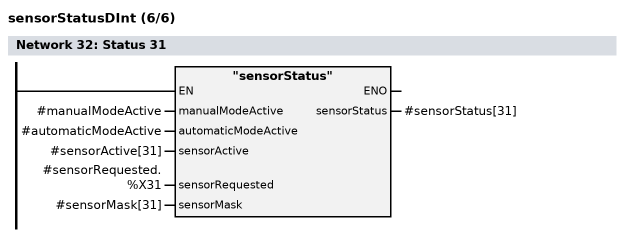
   RUNG wire#powerrail
      "sensorStatus"(manualModeActive := #manualModeActive, automaticModeActive := #automaticModeActive, sensorActive := #sensorActive[31], sensorRequested := #sensorRequested.%X31, sensorMask := #sensorMask[31], sensorStatus => #sensorStatus[31])
   END_RUNG
   // the same network as SCL:
   "sensorStatus"(manualModeActive := #manualModeActive,
                  automaticModeActive := #automaticModeActive,
                  sensorActive := #sensorActive[31],
                  sensorRequested := #sensorRequested.%X31,
                  sensorMask := #sensorMask[31],
                  sensorStatus => #sensorStatus[31]);
END_REGION
END_FUNCTION

FUNCTION "sensorStatus" : Void   // FC36, LAD
{ S7_Optimized_Access := 'TRUE' }
VERSION : 0.1
// stored: AutoNumber true, IsIECCheckEnabled false, SetENOAutomatically false, UDAEnableTagReadback false
   VAR_INPUT
      manualModeActive : Bool;
      automaticModeActive : Bool;
      sensorActive : Bool;
      sensorRequested : Bool;
      sensorMask : Bool;
   END_VAR
   VAR_OUTPUT
      sensorStatus : Int;
   END_VAR
   VAR_TEMP
      localMask : Bool;
   END_VAR
BEGIN

REGION Network 1
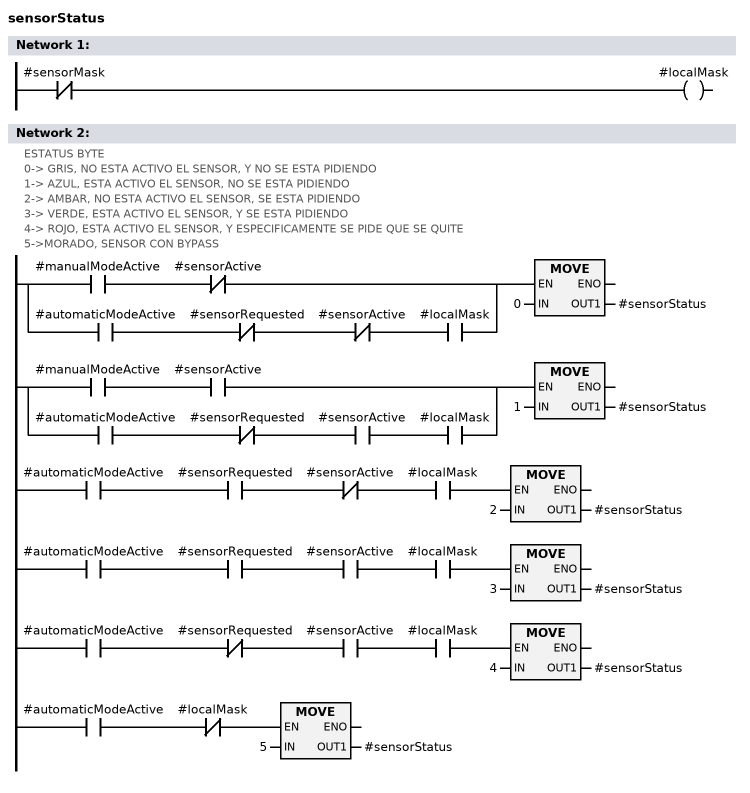
   RUNG wire#powerrail
      I_Contact( #sensorMask )
      Coil( #localMask )
   END_RUNG
   // the same network as SCL:
   #localMask := NOT #sensorMask;
END_REGION

REGION Network 2
   // ESTATUS BYTE
   // 0-> GRIS, NO ESTA ACTIVO EL SENSOR, Y NO SE ESTA PIDIENDO
   // 1-> AZUL, ESTA ACTIVO EL SENSOR, NO SE ESTA PIDIENDO
   // 2-> AMBAR, NO ESTA ACTIVO EL SENSOR, SE ESTA PIDIENDO
   // 3-> VERDE, ESTA ACTIVO EL SENSOR, Y SE ESTA PIDIENDO
   // 4-> ROJO, ESTA ACTIVO EL SENSOR, Y ESPECIFICAMENTE SE PIDE QUE SE QUITE
   // 5->MORADO, SENSOR CON BYPASS
   RUNG wire#powerrail
      Contact( #manualModeActive )
      I_Contact( #sensorActive )
      wire#w1
      Move(in := 0, out1 => #sensorStatus)
   END_RUNG
   RUNG wire#powerrail
      Contact( #automaticModeActive )
      I_Contact( #sensorRequested )
      I_Contact( #sensorActive )
      Contact( #localMask )
   END_RUNG wire#w1
   RUNG wire#powerrail
      Contact( #manualModeActive )
      Contact( #sensorActive )
      wire#w2
      Move(in := 1, out1 => #sensorStatus)
   END_RUNG
   RUNG wire#powerrail
      Contact( #automaticModeActive )
      I_Contact( #sensorRequested )
      Contact( #sensorActive )
      Contact( #localMask )
   END_RUNG wire#w2
   RUNG wire#powerrail
      Contact( #automaticModeActive )
      Contact( #sensorRequested )
      I_Contact( #sensorActive )
      Contact( #localMask )
      Move(in := 2, out1 => #sensorStatus)
   END_RUNG
   RUNG wire#powerrail
      Contact( #automaticModeActive )
      Contact( #sensorRequested )
      Contact( #sensorActive )
      Contact( #localMask )
      Move(in := 3, out1 => #sensorStatus)
   END_RUNG
   RUNG wire#powerrail
      Contact( #automaticModeActive )
      I_Contact( #sensorRequested )
      Contact( #sensorActive )
      Contact( #localMask )
      Move(in := 4, out1 => #sensorStatus)
   END_RUNG
   RUNG wire#powerrail
      Contact( #automaticModeActive )
      I_Contact( #localMask )
      Move(in := 5, out1 => #sensorStatus)
   END_RUNG
   // the same network as SCL:
   IF (#manualModeActive AND NOT #sensorActive) OR (#automaticModeActive AND NOT #sensorRequested AND NOT #sensorActive AND #localMask) THEN
       #sensorStatus := 0;
   END_IF;
   IF (#manualModeActive AND #sensorActive) OR (#automaticModeActive AND NOT #sensorRequested AND #sensorActive AND #localMask) THEN
       #sensorStatus := 1;
   END_IF;
   IF #automaticModeActive AND #sensorRequested AND NOT #sensorActive AND #localMask THEN
       #sensorStatus := 2;
   END_IF;
   IF #automaticModeActive AND #sensorRequested AND #sensorActive AND #localMask THEN
       #sensorStatus := 3;
   END_IF;
   IF #automaticModeActive AND NOT #sensorRequested AND #sensorActive AND #localMask THEN
       #sensorStatus := 4;
   END_IF;
   IF #automaticModeActive AND NOT #localMask THEN #sensorStatus := 5; END_IF;
END_REGION
END_FUNCTION

FUNCTION "cylinderControl" : Void   // FC9, LAD
{ S7_Optimized_Access := 'TRUE' }
VERSION : 0.1
// stored: AutoNumber true, IsIECCheckEnabled false, SetENOAutomatically false, UDAEnableTagReadback false
   VAR_TEMP
      enableCylinders : Bool;
   END_VAR
   VAR_TEMP   // added for the SCL form of the ladder/FBD networks
      _w1 : Bool;
      _w2 : Bool;
   END_VAR
BEGIN

REGION Network 1
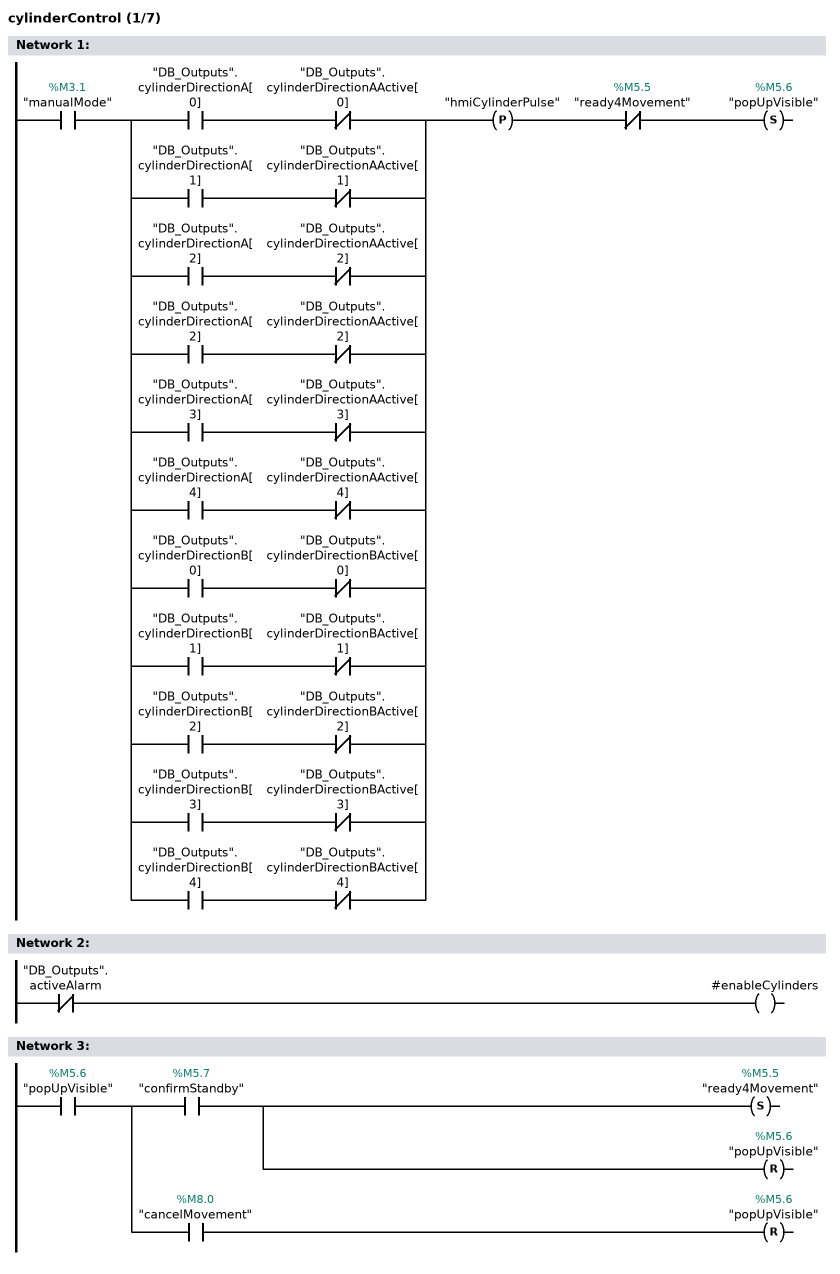
   RUNG wire#powerrail
      Contact( "manualMode" )
      wire#w1
      Contact( "DB_Outputs".cylinderDirectionA[0] )
      I_Contact( "DB_Outputs".cylinderDirectionAActive[0] )
      wire#w2
      P_Trig( "hmiCylinderPulse" )
      I_Contact( "ready4Movement" )
      S_Coil( "popUpVisible" )
   END_RUNG
   RUNG wire#w1
      Contact( "DB_Outputs".cylinderDirectionA[1] )
      I_Contact( "DB_Outputs".cylinderDirectionAActive[1] )
   END_RUNG wire#w2
   RUNG wire#w1
      Contact( "DB_Outputs".cylinderDirectionA[2] )
      I_Contact( "DB_Outputs".cylinderDirectionAActive[2] )
   END_RUNG wire#w2
   RUNG wire#w1
      Contact( "DB_Outputs".cylinderDirectionA[2] )
      I_Contact( "DB_Outputs".cylinderDirectionAActive[2] )
   END_RUNG wire#w2
   RUNG wire#w1
      Contact( "DB_Outputs".cylinderDirectionA[3] )
      I_Contact( "DB_Outputs".cylinderDirectionAActive[3] )
   END_RUNG wire#w2
   RUNG wire#w1
      Contact( "DB_Outputs".cylinderDirectionA[4] )
      I_Contact( "DB_Outputs".cylinderDirectionAActive[4] )
   END_RUNG wire#w2
   RUNG wire#w1
      Contact( "DB_Outputs".cylinderDirectionB[0] )
      I_Contact( "DB_Outputs".cylinderDirectionBActive[0] )
   END_RUNG wire#w2
   RUNG wire#w1
      Contact( "DB_Outputs".cylinderDirectionB[1] )
      I_Contact( "DB_Outputs".cylinderDirectionBActive[1] )
   END_RUNG wire#w2
   RUNG wire#w1
      Contact( "DB_Outputs".cylinderDirectionB[2] )
      I_Contact( "DB_Outputs".cylinderDirectionBActive[2] )
   END_RUNG wire#w2
   RUNG wire#w1
      Contact( "DB_Outputs".cylinderDirectionB[3] )
      I_Contact( "DB_Outputs".cylinderDirectionBActive[3] )
   END_RUNG wire#w2
   RUNG wire#w1
      Contact( "DB_Outputs".cylinderDirectionB[4] )
      I_Contact( "DB_Outputs".cylinderDirectionBActive[4] )
   END_RUNG wire#w2
   // the same network as SCL:
   #_w1 := "manualMode" AND (("DB_Outputs".cylinderDirectionA[0] AND NOT "DB_Outputs".cylinderDirectionAActive[0]) OR ("DB_Outputs".cylinderDirectionA[1] AND NOT "DB_Outputs".cylinderDirectionAActive[1]) OR ("DB_Outputs".cylinderDirectionA[2] AND NOT "DB_Outputs".cylinderDirectionAActive[2]) OR ("DB_Outputs".cylinderDirectionA[2] AND NOT "DB_Outputs".cylinderDirectionAActive[2]) OR ("DB_Outputs".cylinderDirectionA[3] AND NOT "DB_Outputs".cylinderDirectionAActive[3]) OR ("DB_Outputs".cylinderDirectionA[4] AND NOT "DB_Outputs".cylinderDirectionAActive[4]) OR ("DB_Outputs".cylinderDirectionB[0] AND NOT "DB_Outputs".cylinderDirectionBActive[0]) OR ("DB_Outputs".cylinderDirectionB[1] AND NOT "DB_Outputs".cylinderDirectionBActive[1]) OR ("DB_Outputs".cylinderDirectionB[2] AND NOT "DB_Outputs".cylinderDirectionBActive[2]) OR ("DB_Outputs".cylinderDirectionB[3] AND NOT "DB_Outputs".cylinderDirectionBActive[3]) OR ("DB_Outputs".cylinderDirectionB[4] AND NOT "DB_Outputs".cylinderDirectionBActive[4]));
   #_w2 := #_w1 AND NOT "hmiCylinderPulse";   // rising edge
   "hmiCylinderPulse" := #_w1;
   IF #_w2 AND NOT "ready4Movement" THEN "popUpVisible" := TRUE; END_IF;
END_REGION

REGION Network 2
   RUNG wire#powerrail
      I_Contact( "DB_Outputs".activeAlarm )
      Coil( #enableCylinders )
   END_RUNG
   // the same network as SCL:
   #enableCylinders := NOT "DB_Outputs".activeAlarm;
END_REGION

REGION Network 3
   RUNG wire#powerrail
      Contact( "popUpVisible" )
      wire#w1
      Contact( "confirmStandby" )
      wire#w2
      S_Coil( "ready4Movement" )
   END_RUNG
   RUNG wire#w2
      R_Coil( "popUpVisible" )
   END_RUNG
   RUNG wire#w1
      Contact( "cancelMovement" )
      R_Coil( "popUpVisible" )
   END_RUNG
   // the same network as SCL:
   IF "popUpVisible" AND "confirmStandby" THEN "ready4Movement" := TRUE; END_IF;
   #_w1 := "popUpVisible";
   IF "popUpVisible" AND "confirmStandby" THEN "popUpVisible" := FALSE; END_IF;
   IF #_w1 AND "cancelMovement" THEN "popUpVisible" := FALSE; END_IF;
END_REGION

REGION Network 4: EXT CYL 1.- LEFT TOOLING LOCK EXTENDED
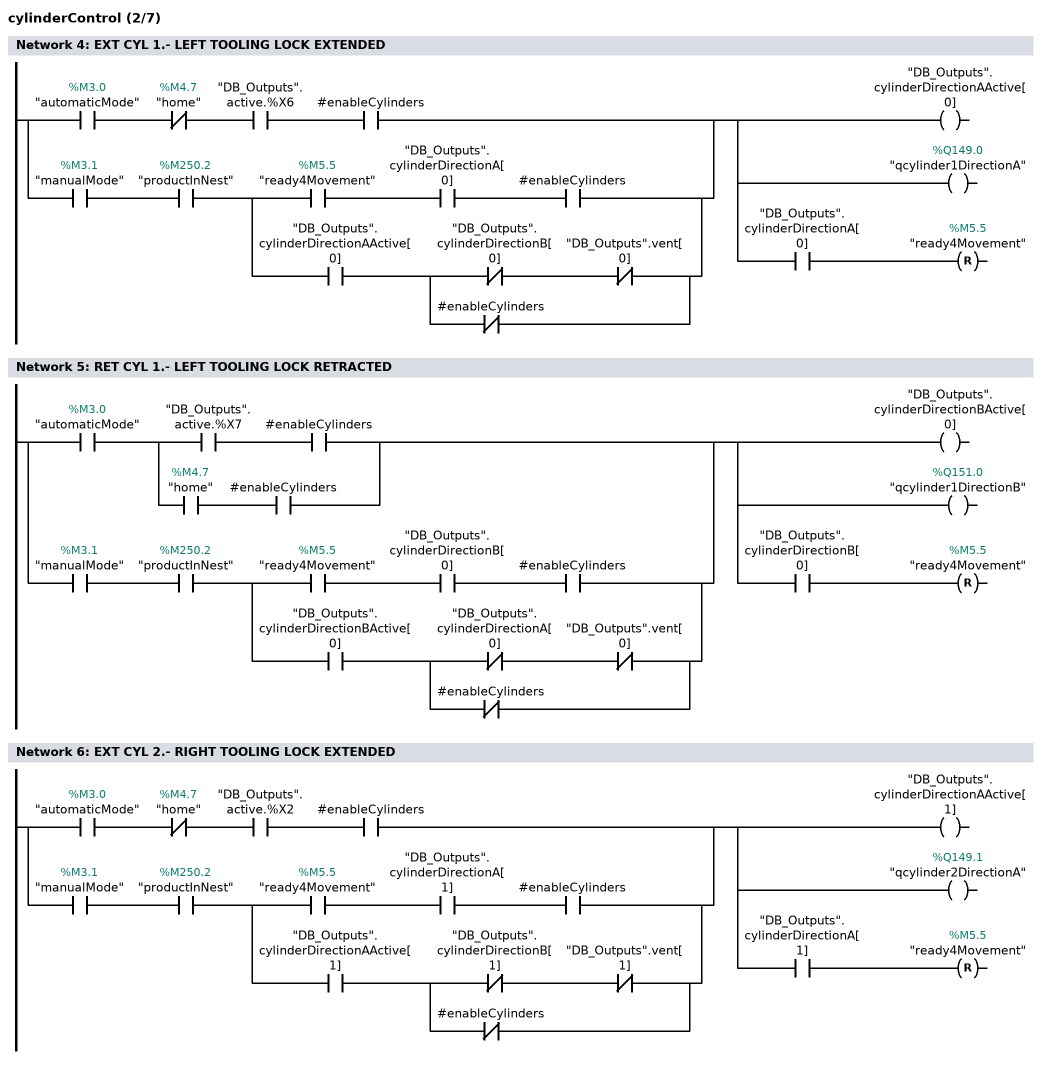
   RUNG wire#powerrail
      Contact( "automaticMode" )
      I_Contact( "home" )
      Contact( "DB_Outputs".active.%X6 )
      Contact( #enableCylinders )
      wire#w1
      Coil( "DB_Outputs".cylinderDirectionAActive[0] )
   END_RUNG
   RUNG wire#powerrail
      Contact( "manualMode" )
      Contact( "productInNest" )
      wire#w2
      Contact( "ready4Movement" )
      Contact( "DB_Outputs".cylinderDirectionA[0] )
      Contact( #enableCylinders )
   END_RUNG wire#w1
   RUNG wire#w2
      Contact( "DB_Outputs".cylinderDirectionAActive[0] )
      wire#w3
      I_Contact( "DB_Outputs".cylinderDirectionB[0] )
      I_Contact( "DB_Outputs".vent[0] )
   END_RUNG wire#w1
   RUNG wire#w3
      I_Contact( #enableCylinders )
   END_RUNG wire#w1
   RUNG wire#w1
      Coil( "qcylinder1DirectionA" )
   END_RUNG
   RUNG wire#w1
      Contact( "DB_Outputs".cylinderDirectionA[0] )
      R_Coil( "ready4Movement" )
   END_RUNG
   // the same network as SCL:
   #_w1 := ("automaticMode" AND NOT "home" AND "DB_Outputs".active.%X6 AND #enableCylinders) OR ("manualMode" AND "productInNest" AND (("ready4Movement" AND "DB_Outputs".cylinderDirectionA[0] AND #enableCylinders) OR ("DB_Outputs".cylinderDirectionAActive[0] AND ((NOT "DB_Outputs".cylinderDirectionB[0] AND NOT "DB_Outputs".vent[0]) OR NOT #enableCylinders))));
   "DB_Outputs".cylinderDirectionAActive[0] := ("automaticMode" AND NOT "home" AND "DB_Outputs".active.%X6 AND #enableCylinders) OR ("manualMode" AND "productInNest" AND (("ready4Movement" AND "DB_Outputs".cylinderDirectionA[0] AND #enableCylinders) OR ("DB_Outputs".cylinderDirectionAActive[0] AND ((NOT "DB_Outputs".cylinderDirectionB[0] AND NOT "DB_Outputs".vent[0]) OR NOT #enableCylinders))));
   "qcylinder1DirectionA" := #_w1;
   IF #_w1 AND "DB_Outputs".cylinderDirectionA[0] THEN "ready4Movement" := FALSE; END_IF;
END_REGION

REGION Network 5: RET CYL 1.- LEFT TOOLING LOCK RETRACTED
   RUNG wire#powerrail
      Contact( "automaticMode" )
      wire#w1
      Contact( "DB_Outputs".active.%X7 )
      Contact( #enableCylinders )
      wire#w2
      Coil( "DB_Outputs".cylinderDirectionBActive[0] )
   END_RUNG
   RUNG wire#w1
      Contact( "home" )
      Contact( #enableCylinders )
   END_RUNG wire#w2
   RUNG wire#powerrail
      Contact( "manualMode" )
      Contact( "productInNest" )
      wire#w3
      Contact( "ready4Movement" )
      Contact( "DB_Outputs".cylinderDirectionB[0] )
      Contact( #enableCylinders )
   END_RUNG wire#w2
   RUNG wire#w3
      Contact( "DB_Outputs".cylinderDirectionBActive[0] )
      wire#w4
      I_Contact( "DB_Outputs".cylinderDirectionA[0] )
      I_Contact( "DB_Outputs".vent[0] )
   END_RUNG wire#w2
   RUNG wire#w4
      I_Contact( #enableCylinders )
   END_RUNG wire#w2
   RUNG wire#w2
      Coil( "qcylinder1DirectionB" )
   END_RUNG
   RUNG wire#w2
      Contact( "DB_Outputs".cylinderDirectionB[0] )
      R_Coil( "ready4Movement" )
   END_RUNG
   // the same network as SCL:
   #_w1 := ("automaticMode" AND (("DB_Outputs".active.%X7 AND #enableCylinders) OR ("home" AND #enableCylinders))) OR ("manualMode" AND "productInNest" AND (("ready4Movement" AND "DB_Outputs".cylinderDirectionB[0] AND #enableCylinders) OR ("DB_Outputs".cylinderDirectionBActive[0] AND ((NOT "DB_Outputs".cylinderDirectionA[0] AND NOT "DB_Outputs".vent[0]) OR NOT #enableCylinders))));
   "DB_Outputs".cylinderDirectionBActive[0] := ("automaticMode" AND (("DB_Outputs".active.%X7 AND #enableCylinders) OR ("home" AND #enableCylinders))) OR ("manualMode" AND "productInNest" AND (("ready4Movement" AND "DB_Outputs".cylinderDirectionB[0] AND #enableCylinders) OR ("DB_Outputs".cylinderDirectionBActive[0] AND ((NOT "DB_Outputs".cylinderDirectionA[0] AND NOT "DB_Outputs".vent[0]) OR NOT #enableCylinders))));
   "qcylinder1DirectionB" := #_w1;
   IF #_w1 AND "DB_Outputs".cylinderDirectionB[0] THEN "ready4Movement" := FALSE; END_IF;
END_REGION

REGION Network 6: EXT CYL 2.- RIGHT TOOLING LOCK EXTENDED
   RUNG wire#powerrail
      Contact( "automaticMode" )
      I_Contact( "home" )
      Contact( "DB_Outputs".active.%X2 )
      Contact( #enableCylinders )
      wire#w1
      Coil( "DB_Outputs".cylinderDirectionAActive[1] )
   END_RUNG
   RUNG wire#powerrail
      Contact( "manualMode" )
      Contact( "productInNest" )
      wire#w2
      Contact( "ready4Movement" )
      Contact( "DB_Outputs".cylinderDirectionA[1] )
      Contact( #enableCylinders )
   END_RUNG wire#w1
   RUNG wire#w2
      Contact( "DB_Outputs".cylinderDirectionAActive[1] )
      wire#w3
      I_Contact( "DB_Outputs".cylinderDirectionB[1] )
      I_Contact( "DB_Outputs".vent[1] )
   END_RUNG wire#w1
   RUNG wire#w3
      I_Contact( #enableCylinders )
   END_RUNG wire#w1
   RUNG wire#w1
      Coil( "qcylinder2DirectionA" )
   END_RUNG
   RUNG wire#w1
      Contact( "DB_Outputs".cylinderDirectionA[1] )
      R_Coil( "ready4Movement" )
   END_RUNG
   // the same network as SCL:
   #_w1 := ("automaticMode" AND NOT "home" AND "DB_Outputs".active.%X2 AND #enableCylinders) OR ("manualMode" AND "productInNest" AND (("ready4Movement" AND "DB_Outputs".cylinderDirectionA[1] AND #enableCylinders) OR ("DB_Outputs".cylinderDirectionAActive[1] AND ((NOT "DB_Outputs".cylinderDirectionB[1] AND NOT "DB_Outputs".vent[1]) OR NOT #enableCylinders))));
   "DB_Outputs".cylinderDirectionAActive[1] := ("automaticMode" AND NOT "home" AND "DB_Outputs".active.%X2 AND #enableCylinders) OR ("manualMode" AND "productInNest" AND (("ready4Movement" AND "DB_Outputs".cylinderDirectionA[1] AND #enableCylinders) OR ("DB_Outputs".cylinderDirectionAActive[1] AND ((NOT "DB_Outputs".cylinderDirectionB[1] AND NOT "DB_Outputs".vent[1]) OR NOT #enableCylinders))));
   "qcylinder2DirectionA" := #_w1;
   IF #_w1 AND "DB_Outputs".cylinderDirectionA[1] THEN "ready4Movement" := FALSE; END_IF;
END_REGION

REGION Network 7: RET CYL 2.- RIGHT TOOLING LOCK RETRACTED
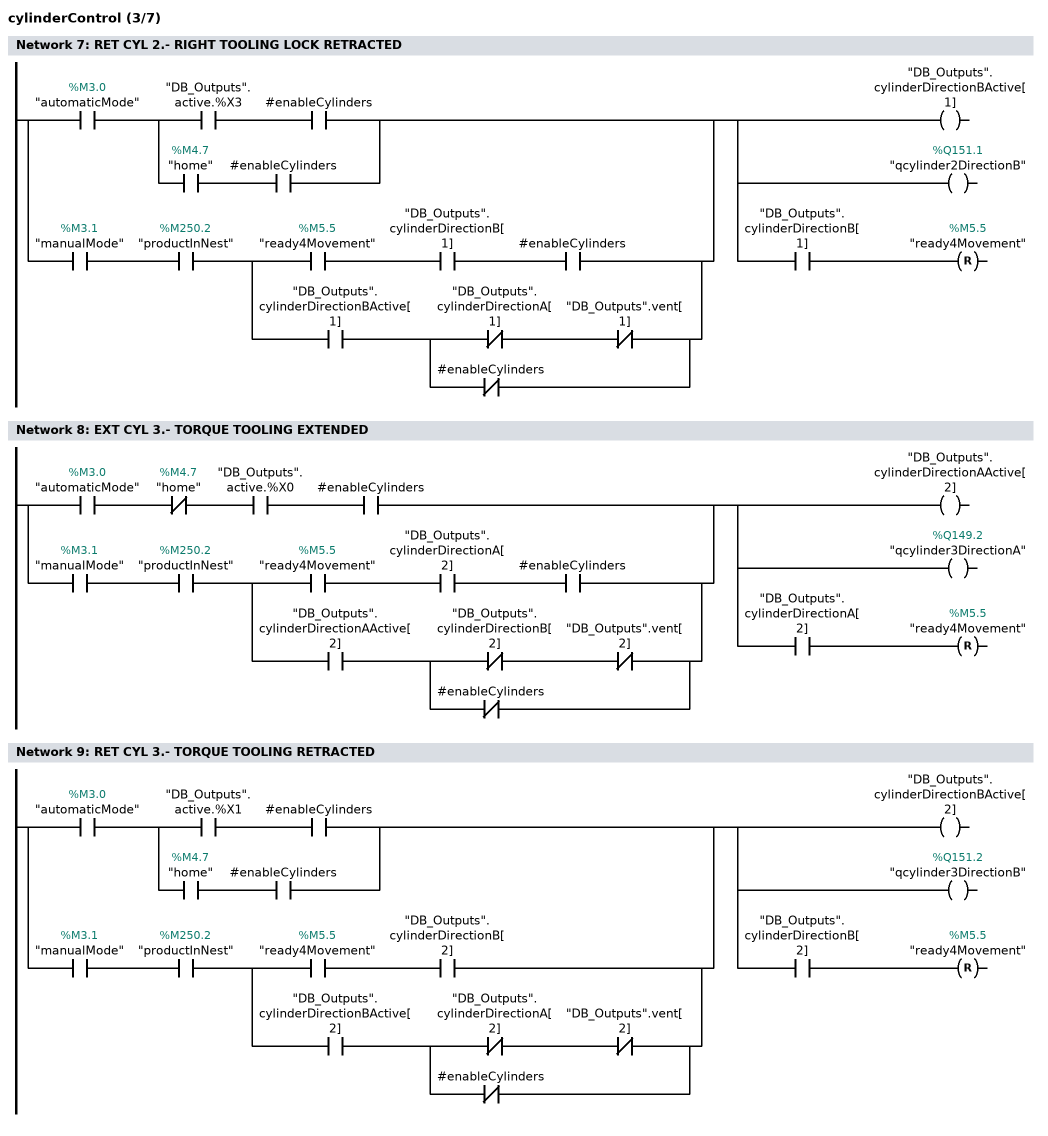
   RUNG wire#powerrail
      Contact( "automaticMode" )
      wire#w1
      Contact( "DB_Outputs".active.%X3 )
      Contact( #enableCylinders )
      wire#w2
      Coil( "DB_Outputs".cylinderDirectionBActive[1] )
   END_RUNG
   RUNG wire#w1
      Contact( "home" )
      Contact( #enableCylinders )
   END_RUNG wire#w2
   RUNG wire#powerrail
      Contact( "manualMode" )
      Contact( "productInNest" )
      wire#w3
      Contact( "ready4Movement" )
      Contact( "DB_Outputs".cylinderDirectionB[1] )
      Contact( #enableCylinders )
   END_RUNG wire#w2
   RUNG wire#w3
      Contact( "DB_Outputs".cylinderDirectionBActive[1] )
      wire#w4
      I_Contact( "DB_Outputs".cylinderDirectionA[1] )
      I_Contact( "DB_Outputs".vent[1] )
   END_RUNG wire#w2
   RUNG wire#w4
      I_Contact( #enableCylinders )
   END_RUNG wire#w2
   RUNG wire#w2
      Coil( "qcylinder2DirectionB" )
   END_RUNG
   RUNG wire#w2
      Contact( "DB_Outputs".cylinderDirectionB[1] )
      R_Coil( "ready4Movement" )
   END_RUNG
   // the same network as SCL:
   #_w1 := ("automaticMode" AND (("DB_Outputs".active.%X3 AND #enableCylinders) OR ("home" AND #enableCylinders))) OR ("manualMode" AND "productInNest" AND (("ready4Movement" AND "DB_Outputs".cylinderDirectionB[1] AND #enableCylinders) OR ("DB_Outputs".cylinderDirectionBActive[1] AND ((NOT "DB_Outputs".cylinderDirectionA[1] AND NOT "DB_Outputs".vent[1]) OR NOT #enableCylinders))));
   "DB_Outputs".cylinderDirectionBActive[1] := ("automaticMode" AND (("DB_Outputs".active.%X3 AND #enableCylinders) OR ("home" AND #enableCylinders))) OR ("manualMode" AND "productInNest" AND (("ready4Movement" AND "DB_Outputs".cylinderDirectionB[1] AND #enableCylinders) OR ("DB_Outputs".cylinderDirectionBActive[1] AND ((NOT "DB_Outputs".cylinderDirectionA[1] AND NOT "DB_Outputs".vent[1]) OR NOT #enableCylinders))));
   "qcylinder2DirectionB" := #_w1;
   IF #_w1 AND "DB_Outputs".cylinderDirectionB[1] THEN "ready4Movement" := FALSE; END_IF;
END_REGION

REGION Network 8: EXT CYL 3.- TORQUE TOOLING EXTENDED
   RUNG wire#powerrail
      Contact( "automaticMode" )
      I_Contact( "home" )
      Contact( "DB_Outputs".active.%X0 )
      Contact( #enableCylinders )
      wire#w1
      Coil( "DB_Outputs".cylinderDirectionAActive[2] )
   END_RUNG
   RUNG wire#powerrail
      Contact( "manualMode" )
      Contact( "productInNest" )
      wire#w2
      Contact( "ready4Movement" )
      Contact( "DB_Outputs".cylinderDirectionA[2] )
      Contact( #enableCylinders )
   END_RUNG wire#w1
   RUNG wire#w2
      Contact( "DB_Outputs".cylinderDirectionAActive[2] )
      wire#w3
      I_Contact( "DB_Outputs".cylinderDirectionB[2] )
      I_Contact( "DB_Outputs".vent[2] )
   END_RUNG wire#w1
   RUNG wire#w3
      I_Contact( #enableCylinders )
   END_RUNG wire#w1
   RUNG wire#w1
      Coil( "qcylinder3DirectionA" )
   END_RUNG
   RUNG wire#w1
      Contact( "DB_Outputs".cylinderDirectionA[2] )
      R_Coil( "ready4Movement" )
   END_RUNG
   // the same network as SCL:
   #_w1 := ("automaticMode" AND NOT "home" AND "DB_Outputs".active.%X0 AND #enableCylinders) OR ("manualMode" AND "productInNest" AND (("ready4Movement" AND "DB_Outputs".cylinderDirectionA[2] AND #enableCylinders) OR ("DB_Outputs".cylinderDirectionAActive[2] AND ((NOT "DB_Outputs".cylinderDirectionB[2] AND NOT "DB_Outputs".vent[2]) OR NOT #enableCylinders))));
   "DB_Outputs".cylinderDirectionAActive[2] := ("automaticMode" AND NOT "home" AND "DB_Outputs".active.%X0 AND #enableCylinders) OR ("manualMode" AND "productInNest" AND (("ready4Movement" AND "DB_Outputs".cylinderDirectionA[2] AND #enableCylinders) OR ("DB_Outputs".cylinderDirectionAActive[2] AND ((NOT "DB_Outputs".cylinderDirectionB[2] AND NOT "DB_Outputs".vent[2]) OR NOT #enableCylinders))));
   "qcylinder3DirectionA" := #_w1;
   IF #_w1 AND "DB_Outputs".cylinderDirectionA[2] THEN "ready4Movement" := FALSE; END_IF;
END_REGION

REGION Network 9: RET CYL 3.- TORQUE TOOLING RETRACTED
   RUNG wire#powerrail
      Contact( "automaticMode" )
      wire#w1
      Contact( "DB_Outputs".active.%X1 )
      Contact( #enableCylinders )
      wire#w2
      Coil( "DB_Outputs".cylinderDirectionBActive[2] )
   END_RUNG
   RUNG wire#w1
      Contact( "home" )
      Contact( #enableCylinders )
   END_RUNG wire#w2
   RUNG wire#powerrail
      Contact( "manualMode" )
      Contact( "productInNest" )
      wire#w3
      Contact( "ready4Movement" )
      Contact( "DB_Outputs".cylinderDirectionB[2] )
   END_RUNG wire#w2
   RUNG wire#w3
      Contact( "DB_Outputs".cylinderDirectionBActive[2] )
      wire#w4
      I_Contact( "DB_Outputs".cylinderDirectionA[2] )
      I_Contact( "DB_Outputs".vent[2] )
   END_RUNG wire#w2
   RUNG wire#w4
      I_Contact( #enableCylinders )
   END_RUNG wire#w2
   RUNG wire#w2
      Coil( "qcylinder3DirectionB" )
   END_RUNG
   RUNG wire#w2
      Contact( "DB_Outputs".cylinderDirectionB[2] )
      R_Coil( "ready4Movement" )
   END_RUNG
   // the same network as SCL:
   #_w1 := ("automaticMode" AND (("DB_Outputs".active.%X1 AND #enableCylinders) OR ("home" AND #enableCylinders))) OR ("manualMode" AND "productInNest" AND (("ready4Movement" AND "DB_Outputs".cylinderDirectionB[2]) OR ("DB_Outputs".cylinderDirectionBActive[2] AND ((NOT "DB_Outputs".cylinderDirectionA[2] AND NOT "DB_Outputs".vent[2]) OR NOT #enableCylinders))));
   "DB_Outputs".cylinderDirectionBActive[2] := ("automaticMode" AND (("DB_Outputs".active.%X1 AND #enableCylinders) OR ("home" AND #enableCylinders))) OR ("manualMode" AND "productInNest" AND (("ready4Movement" AND "DB_Outputs".cylinderDirectionB[2]) OR ("DB_Outputs".cylinderDirectionBActive[2] AND ((NOT "DB_Outputs".cylinderDirectionA[2] AND NOT "DB_Outputs".vent[2]) OR NOT #enableCylinders))));
   "qcylinder3DirectionB" := #_w1;
   IF #_w1 AND "DB_Outputs".cylinderDirectionB[2] THEN "ready4Movement" := FALSE; END_IF;
END_REGION

REGION Network 10: EXT CYL 4.- RIGTH ROD INSERTION EXTENDED
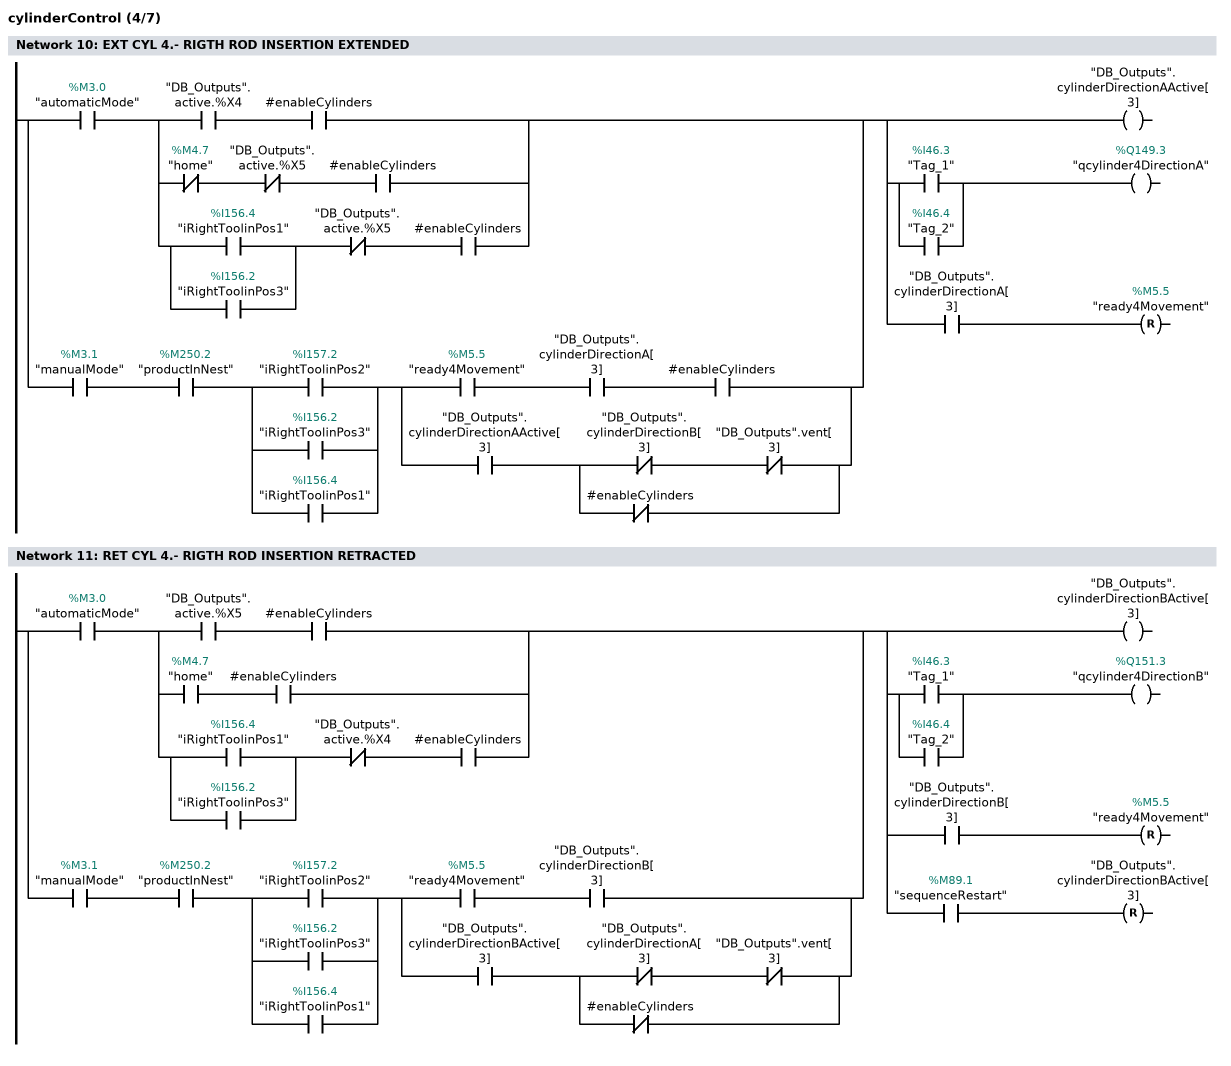
   RUNG wire#powerrail
      Contact( "automaticMode" )
      wire#w1
      Contact( "DB_Outputs".active.%X4 )
      Contact( #enableCylinders )
      wire#w2
      Coil( "DB_Outputs".cylinderDirectionAActive[3] )
   END_RUNG
   RUNG wire#w1
      I_Contact( "home" )
      I_Contact( "DB_Outputs".active.%X5 )
      Contact( #enableCylinders )
   END_RUNG wire#w2
   RUNG wire#w1
      Contact( "iRightToolinPos1" )
      wire#w3
      I_Contact( "DB_Outputs".active.%X5 )
      Contact( #enableCylinders )
   END_RUNG wire#w2
   RUNG wire#w1
      Contact( "iRightToolinPos3" )
   END_RUNG wire#w3
   RUNG wire#powerrail
      Contact( "manualMode" )
      Contact( "productInNest" )
      wire#w4
      Contact( "iRightToolinPos2" )
      wire#w5
      Contact( "ready4Movement" )
      Contact( "DB_Outputs".cylinderDirectionA[3] )
      Contact( #enableCylinders )
   END_RUNG wire#w2
   RUNG wire#w4
      Contact( "iRightToolinPos3" )
   END_RUNG wire#w5
   RUNG wire#w4
      Contact( "iRightToolinPos1" )
   END_RUNG wire#w5
   RUNG wire#w5
      Contact( "DB_Outputs".cylinderDirectionAActive[3] )
      wire#w6
      I_Contact( "DB_Outputs".cylinderDirectionB[3] )
      I_Contact( "DB_Outputs".vent[3] )
   END_RUNG wire#w2
   RUNG wire#w6
      I_Contact( #enableCylinders )
   END_RUNG wire#w2
   RUNG wire#w2
      Contact( "Tag_1" )
      wire#w7
      Coil( "qcylinder4DirectionA" )
   END_RUNG
   RUNG wire#w2
      Contact( "Tag_2" )
   END_RUNG wire#w7
   RUNG wire#w2
      Contact( "DB_Outputs".cylinderDirectionA[3] )
      R_Coil( "ready4Movement" )
   END_RUNG
   // the same network as SCL:
   #_w1 := ("automaticMode" AND (("DB_Outputs".active.%X4 AND #enableCylinders) OR (NOT "home" AND NOT "DB_Outputs".active.%X5 AND #enableCylinders) OR (("iRightToolinPos1" OR "iRightToolinPos3") AND NOT "DB_Outputs".active.%X5 AND #enableCylinders))) OR ("manualMode" AND "productInNest" AND ("iRightToolinPos2" OR "iRightToolinPos3" OR "iRightToolinPos1") AND (("ready4Movement" AND "DB_Outputs".cylinderDirectionA[3] AND #enableCylinders) OR ("DB_Outputs".cylinderDirectionAActive[3] AND ((NOT "DB_Outputs".cylinderDirectionB[3] AND NOT "DB_Outputs".vent[3]) OR NOT #enableCylinders))));
   "DB_Outputs".cylinderDirectionAActive[3] := ("automaticMode" AND (("DB_Outputs".active.%X4 AND #enableCylinders) OR (NOT "home" AND NOT "DB_Outputs".active.%X5 AND #enableCylinders) OR (("iRightToolinPos1" OR "iRightToolinPos3") AND NOT "DB_Outputs".active.%X5 AND #enableCylinders))) OR ("manualMode" AND "productInNest" AND ("iRightToolinPos2" OR "iRightToolinPos3" OR "iRightToolinPos1") AND (("ready4Movement" AND "DB_Outputs".cylinderDirectionA[3] AND #enableCylinders) OR ("DB_Outputs".cylinderDirectionAActive[3] AND ((NOT "DB_Outputs".cylinderDirectionB[3] AND NOT "DB_Outputs".vent[3]) OR NOT #enableCylinders))));
   "qcylinder4DirectionA" := #_w1 AND ("Tag_1" OR "Tag_2");
   IF #_w1 AND "DB_Outputs".cylinderDirectionA[3] THEN "ready4Movement" := FALSE; END_IF;
END_REGION

REGION Network 11: RET CYL 4.- RIGTH ROD INSERTION RETRACTED
   RUNG wire#powerrail
      Contact( "automaticMode" )
      wire#w1
      Contact( "DB_Outputs".active.%X5 )
      Contact( #enableCylinders )
      wire#w2
      Coil( "DB_Outputs".cylinderDirectionBActive[3] )
   END_RUNG
   RUNG wire#w1
      Contact( "home" )
      Contact( #enableCylinders )
   END_RUNG wire#w2
   RUNG wire#w1
      Contact( "iRightToolinPos1" )
      wire#w3
      I_Contact( "DB_Outputs".active.%X4 )
      Contact( #enableCylinders )
   END_RUNG wire#w2
   RUNG wire#w1
      Contact( "iRightToolinPos3" )
   END_RUNG wire#w3
   RUNG wire#powerrail
      Contact( "manualMode" )
      Contact( "productInNest" )
      wire#w4
      Contact( "iRightToolinPos2" )
      wire#w5
      Contact( "ready4Movement" )
      Contact( "DB_Outputs".cylinderDirectionB[3] )
   END_RUNG wire#w2
   RUNG wire#w4
      Contact( "iRightToolinPos3" )
   END_RUNG wire#w5
   RUNG wire#w4
      Contact( "iRightToolinPos1" )
   END_RUNG wire#w5
   RUNG wire#w5
      Contact( "DB_Outputs".cylinderDirectionBActive[3] )
      wire#w6
      I_Contact( "DB_Outputs".cylinderDirectionA[3] )
      I_Contact( "DB_Outputs".vent[3] )
   END_RUNG wire#w2
   RUNG wire#w6
      I_Contact( #enableCylinders )
   END_RUNG wire#w2
   RUNG wire#w2
      Contact( "Tag_1" )
      wire#w7
      Coil( "qcylinder4DirectionB" )
   END_RUNG
   RUNG wire#w2
      Contact( "Tag_2" )
   END_RUNG wire#w7
   RUNG wire#w2
      Contact( "DB_Outputs".cylinderDirectionB[3] )
      R_Coil( "ready4Movement" )
   END_RUNG
   RUNG wire#w2
      Contact( "sequenceRestart" )
      R_Coil( "DB_Outputs".cylinderDirectionBActive[3] )
   END_RUNG
   // the same network as SCL:
   #_w1 := ("automaticMode" AND (("DB_Outputs".active.%X5 AND #enableCylinders) OR ("home" AND #enableCylinders) OR (("iRightToolinPos1" OR "iRightToolinPos3") AND NOT "DB_Outputs".active.%X4 AND #enableCylinders))) OR ("manualMode" AND "productInNest" AND ("iRightToolinPos2" OR "iRightToolinPos3" OR "iRightToolinPos1") AND (("ready4Movement" AND "DB_Outputs".cylinderDirectionB[3]) OR ("DB_Outputs".cylinderDirectionBActive[3] AND ((NOT "DB_Outputs".cylinderDirectionA[3] AND NOT "DB_Outputs".vent[3]) OR NOT #enableCylinders))));
   "DB_Outputs".cylinderDirectionBActive[3] := ("automaticMode" AND (("DB_Outputs".active.%X5 AND #enableCylinders) OR ("home" AND #enableCylinders) OR (("iRightToolinPos1" OR "iRightToolinPos3") AND NOT "DB_Outputs".active.%X4 AND #enableCylinders))) OR ("manualMode" AND "productInNest" AND ("iRightToolinPos2" OR "iRightToolinPos3" OR "iRightToolinPos1") AND (("ready4Movement" AND "DB_Outputs".cylinderDirectionB[3]) OR ("DB_Outputs".cylinderDirectionBActive[3] AND ((NOT "DB_Outputs".cylinderDirectionA[3] AND NOT "DB_Outputs".vent[3]) OR NOT #enableCylinders))));
   "qcylinder4DirectionB" := #_w1 AND ("Tag_1" OR "Tag_2");
   IF #_w1 AND "DB_Outputs".cylinderDirectionB[3] THEN "ready4Movement" := FALSE; END_IF;
   IF #_w1 AND "sequenceRestart" THEN "DB_Outputs".cylinderDirectionBActive[3] := FALSE; END_IF;
END_REGION

REGION Network 12: EXT CYL 5.- LEFT WASHER/ROD INSERTION EXTENDED
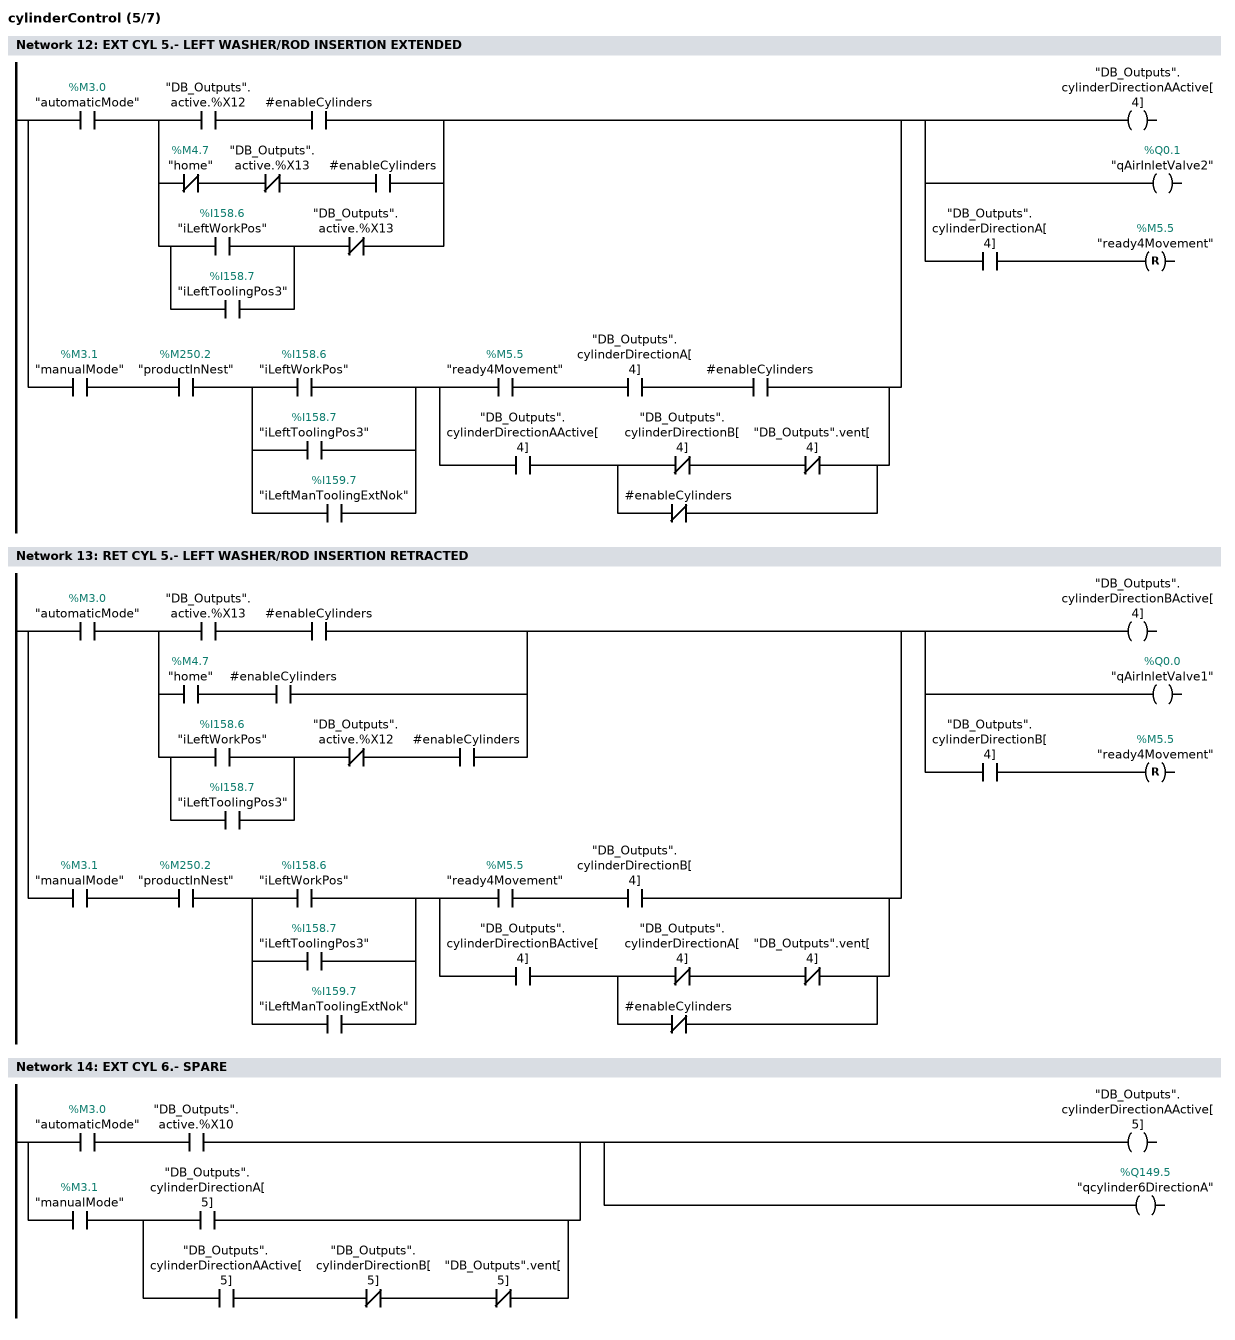
   RUNG wire#powerrail
      Contact( "automaticMode" )
      wire#w1
      Contact( "DB_Outputs".active.%X12 )
      Contact( #enableCylinders )
      wire#w2
      Coil( "DB_Outputs".cylinderDirectionAActive[4] )
   END_RUNG
   RUNG wire#w1
      I_Contact( "home" )
      I_Contact( "DB_Outputs".active.%X13 )
      Contact( #enableCylinders )
   END_RUNG wire#w2
   RUNG wire#w1
      Contact( "iLeftWorkPos" )
      wire#w3
      I_Contact( "DB_Outputs".active.%X13 )
   END_RUNG wire#w2
   RUNG wire#w1
      Contact( "iLeftToolingPos3" )
   END_RUNG wire#w3
   RUNG wire#powerrail
      Contact( "manualMode" )
      Contact( "productInNest" )
      wire#w4
      Contact( "iLeftWorkPos" )
      wire#w5
      Contact( "ready4Movement" )
      Contact( "DB_Outputs".cylinderDirectionA[4] )
      Contact( #enableCylinders )
   END_RUNG wire#w2
   RUNG wire#w4
      Contact( "iLeftToolingPos3" )
   END_RUNG wire#w5
   RUNG wire#w4
      Contact( "iLeftManToolingExtNok" )
   END_RUNG wire#w5
   RUNG wire#w5
      Contact( "DB_Outputs".cylinderDirectionAActive[4] )
      wire#w6
      I_Contact( "DB_Outputs".cylinderDirectionB[4] )
      I_Contact( "DB_Outputs".vent[4] )
   END_RUNG wire#w2
   RUNG wire#w6
      I_Contact( #enableCylinders )
   END_RUNG wire#w2
   RUNG wire#w2
      Coil( "qAirInletValve2" )
   END_RUNG
   RUNG wire#w2
      Contact( "DB_Outputs".cylinderDirectionA[4] )
      R_Coil( "ready4Movement" )
   END_RUNG
   // the same network as SCL:
   #_w1 := ("automaticMode" AND (("DB_Outputs".active.%X12 AND #enableCylinders) OR (NOT "home" AND NOT "DB_Outputs".active.%X13 AND #enableCylinders) OR (("iLeftWorkPos" OR "iLeftToolingPos3") AND NOT "DB_Outputs".active.%X13))) OR ("manualMode" AND "productInNest" AND ("iLeftWorkPos" OR "iLeftToolingPos3" OR "iLeftManToolingExtNok") AND (("ready4Movement" AND "DB_Outputs".cylinderDirectionA[4] AND #enableCylinders) OR ("DB_Outputs".cylinderDirectionAActive[4] AND ((NOT "DB_Outputs".cylinderDirectionB[4] AND NOT "DB_Outputs".vent[4]) OR NOT #enableCylinders))));
   "DB_Outputs".cylinderDirectionAActive[4] := ("automaticMode" AND (("DB_Outputs".active.%X12 AND #enableCylinders) OR (NOT "home" AND NOT "DB_Outputs".active.%X13 AND #enableCylinders) OR (("iLeftWorkPos" OR "iLeftToolingPos3") AND NOT "DB_Outputs".active.%X13))) OR ("manualMode" AND "productInNest" AND ("iLeftWorkPos" OR "iLeftToolingPos3" OR "iLeftManToolingExtNok") AND (("ready4Movement" AND "DB_Outputs".cylinderDirectionA[4] AND #enableCylinders) OR ("DB_Outputs".cylinderDirectionAActive[4] AND ((NOT "DB_Outputs".cylinderDirectionB[4] AND NOT "DB_Outputs".vent[4]) OR NOT #enableCylinders))));
   "qAirInletValve2" := #_w1;
   IF #_w1 AND "DB_Outputs".cylinderDirectionA[4] THEN "ready4Movement" := FALSE; END_IF;
END_REGION

REGION Network 13: RET CYL 5.- LEFT WASHER/ROD INSERTION RETRACTED
   RUNG wire#powerrail
      Contact( "automaticMode" )
      wire#w1
      Contact( "DB_Outputs".active.%X13 )
      Contact( #enableCylinders )
      wire#w2
      Coil( "DB_Outputs".cylinderDirectionBActive[4] )
   END_RUNG
   RUNG wire#w1
      Contact( "home" )
      Contact( #enableCylinders )
   END_RUNG wire#w2
   RUNG wire#w1
      Contact( "iLeftWorkPos" )
      wire#w3
      I_Contact( "DB_Outputs".active.%X12 )
      Contact( #enableCylinders )
   END_RUNG wire#w2
   RUNG wire#w1
      Contact( "iLeftToolingPos3" )
   END_RUNG wire#w3
   RUNG wire#powerrail
      Contact( "manualMode" )
      Contact( "productInNest" )
      wire#w4
      Contact( "iLeftWorkPos" )
      wire#w5
      Contact( "ready4Movement" )
      Contact( "DB_Outputs".cylinderDirectionB[4] )
   END_RUNG wire#w2
   RUNG wire#w4
      Contact( "iLeftToolingPos3" )
   END_RUNG wire#w5
   RUNG wire#w4
      Contact( "iLeftManToolingExtNok" )
   END_RUNG wire#w5
   RUNG wire#w5
      Contact( "DB_Outputs".cylinderDirectionBActive[4] )
      wire#w6
      I_Contact( "DB_Outputs".cylinderDirectionA[4] )
      I_Contact( "DB_Outputs".vent[4] )
   END_RUNG wire#w2
   RUNG wire#w6
      I_Contact( #enableCylinders )
   END_RUNG wire#w2
   RUNG wire#w2
      Coil( "qAirInletValve1" )
   END_RUNG
   RUNG wire#w2
      Contact( "DB_Outputs".cylinderDirectionB[4] )
      R_Coil( "ready4Movement" )
   END_RUNG
   // the same network as SCL:
   #_w1 := ("automaticMode" AND (("DB_Outputs".active.%X13 AND #enableCylinders) OR ("home" AND #enableCylinders) OR (("iLeftWorkPos" OR "iLeftToolingPos3") AND NOT "DB_Outputs".active.%X12 AND #enableCylinders))) OR ("manualMode" AND "productInNest" AND ("iLeftWorkPos" OR "iLeftToolingPos3" OR "iLeftManToolingExtNok") AND (("ready4Movement" AND "DB_Outputs".cylinderDirectionB[4]) OR ("DB_Outputs".cylinderDirectionBActive[4] AND ((NOT "DB_Outputs".cylinderDirectionA[4] AND NOT "DB_Outputs".vent[4]) OR NOT #enableCylinders))));
   "DB_Outputs".cylinderDirectionBActive[4] := ("automaticMode" AND (("DB_Outputs".active.%X13 AND #enableCylinders) OR ("home" AND #enableCylinders) OR (("iLeftWorkPos" OR "iLeftToolingPos3") AND NOT "DB_Outputs".active.%X12 AND #enableCylinders))) OR ("manualMode" AND "productInNest" AND ("iLeftWorkPos" OR "iLeftToolingPos3" OR "iLeftManToolingExtNok") AND (("ready4Movement" AND "DB_Outputs".cylinderDirectionB[4]) OR ("DB_Outputs".cylinderDirectionBActive[4] AND ((NOT "DB_Outputs".cylinderDirectionA[4] AND NOT "DB_Outputs".vent[4]) OR NOT #enableCylinders))));
   "qAirInletValve1" := #_w1;
   IF #_w1 AND "DB_Outputs".cylinderDirectionB[4] THEN "ready4Movement" := FALSE; END_IF;
END_REGION

REGION Network 14: EXT CYL 6.- SPARE
   RUNG wire#powerrail
      Contact( "automaticMode" )
      Contact( "DB_Outputs".active.%X10 )
      wire#w1
      Coil( "DB_Outputs".cylinderDirectionAActive[5] )
   END_RUNG
   RUNG wire#powerrail
      Contact( "manualMode" )
      wire#w2
      Contact( "DB_Outputs".cylinderDirectionA[5] )
   END_RUNG wire#w1
   RUNG wire#w2
      Contact( "DB_Outputs".cylinderDirectionAActive[5] )
      I_Contact( "DB_Outputs".cylinderDirectionB[5] )
      I_Contact( "DB_Outputs".vent[5] )
   END_RUNG wire#w1
   RUNG wire#w1
      Coil( "qcylinder6DirectionA" )
   END_RUNG
   // the same network as SCL:
   #_w1 := ("automaticMode" AND "DB_Outputs".active.%X10) OR ("manualMode" AND ("DB_Outputs".cylinderDirectionA[5] OR ("DB_Outputs".cylinderDirectionAActive[5] AND NOT "DB_Outputs".cylinderDirectionB[5] AND NOT "DB_Outputs".vent[5])));
   "DB_Outputs".cylinderDirectionAActive[5] := ("automaticMode" AND "DB_Outputs".active.%X10) OR ("manualMode" AND ("DB_Outputs".cylinderDirectionA[5] OR ("DB_Outputs".cylinderDirectionAActive[5] AND NOT "DB_Outputs".cylinderDirectionB[5] AND NOT "DB_Outputs".vent[5])));
   "qcylinder6DirectionA" := #_w1;
END_REGION

REGION Network 15: RET CYL 6.- SPARE
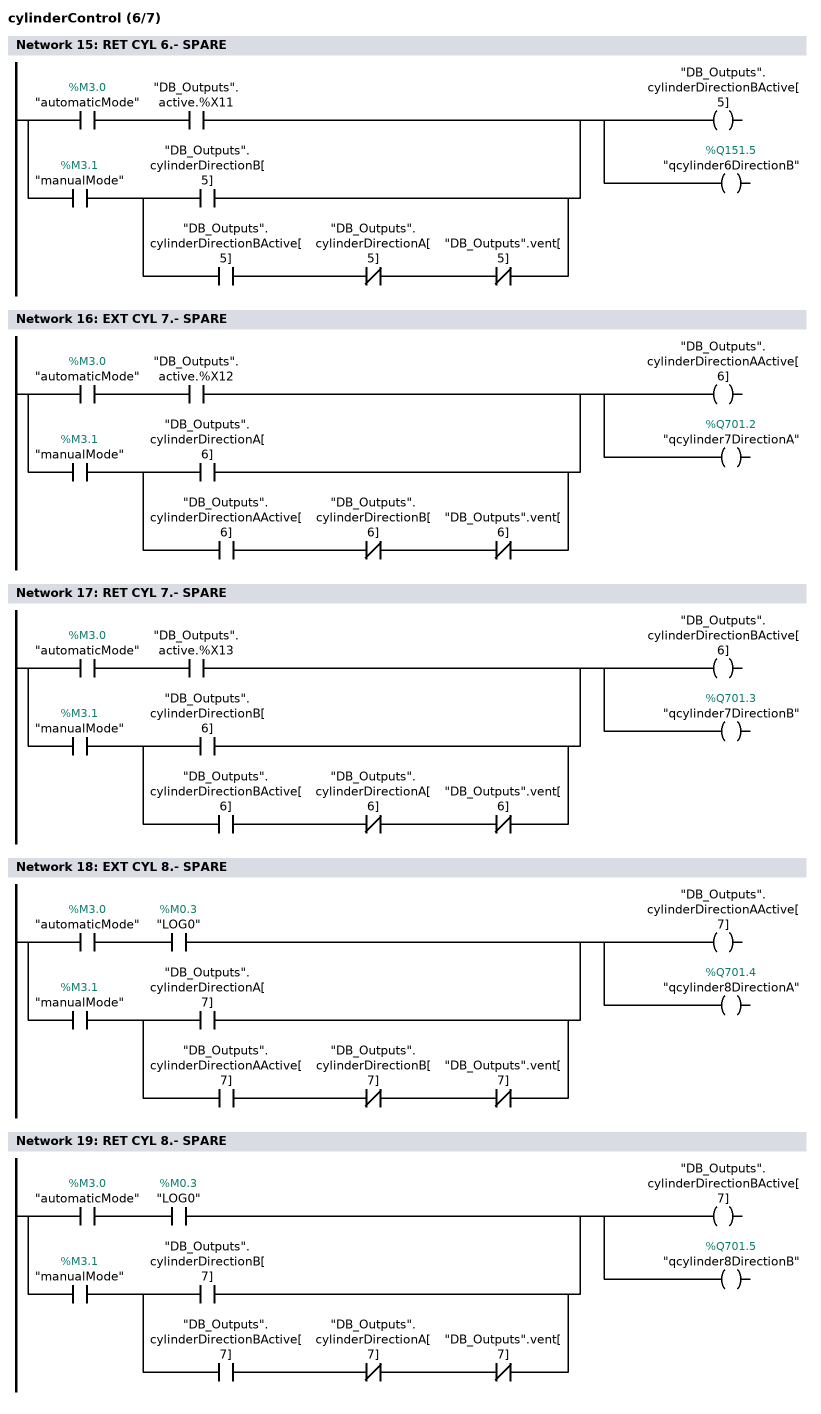
   RUNG wire#powerrail
      Contact( "automaticMode" )
      Contact( "DB_Outputs".active.%X11 )
      wire#w1
      Coil( "DB_Outputs".cylinderDirectionBActive[5] )
   END_RUNG
   RUNG wire#powerrail
      Contact( "manualMode" )
      wire#w2
      Contact( "DB_Outputs".cylinderDirectionB[5] )
   END_RUNG wire#w1
   RUNG wire#w2
      Contact( "DB_Outputs".cylinderDirectionBActive[5] )
      I_Contact( "DB_Outputs".cylinderDirectionA[5] )
      I_Contact( "DB_Outputs".vent[5] )
   END_RUNG wire#w1
   RUNG wire#w1
      Coil( "qcylinder6DirectionB" )
   END_RUNG
   // the same network as SCL:
   #_w1 := ("automaticMode" AND "DB_Outputs".active.%X11) OR ("manualMode" AND ("DB_Outputs".cylinderDirectionB[5] OR ("DB_Outputs".cylinderDirectionBActive[5] AND NOT "DB_Outputs".cylinderDirectionA[5] AND NOT "DB_Outputs".vent[5])));
   "DB_Outputs".cylinderDirectionBActive[5] := ("automaticMode" AND "DB_Outputs".active.%X11) OR ("manualMode" AND ("DB_Outputs".cylinderDirectionB[5] OR ("DB_Outputs".cylinderDirectionBActive[5] AND NOT "DB_Outputs".cylinderDirectionA[5] AND NOT "DB_Outputs".vent[5])));
   "qcylinder6DirectionB" := #_w1;
END_REGION

REGION Network 16: EXT CYL 7.- SPARE
   RUNG wire#powerrail
      Contact( "automaticMode" )
      Contact( "DB_Outputs".active.%X12 )
      wire#w1
      Coil( "DB_Outputs".cylinderDirectionAActive[6] )
   END_RUNG
   RUNG wire#powerrail
      Contact( "manualMode" )
      wire#w2
      Contact( "DB_Outputs".cylinderDirectionA[6] )
   END_RUNG wire#w1
   RUNG wire#w2
      Contact( "DB_Outputs".cylinderDirectionAActive[6] )
      I_Contact( "DB_Outputs".cylinderDirectionB[6] )
      I_Contact( "DB_Outputs".vent[6] )
   END_RUNG wire#w1
   RUNG wire#w1
      Coil( "qcylinder7DirectionA" )
   END_RUNG
   // the same network as SCL:
   #_w1 := ("automaticMode" AND "DB_Outputs".active.%X12) OR ("manualMode" AND ("DB_Outputs".cylinderDirectionA[6] OR ("DB_Outputs".cylinderDirectionAActive[6] AND NOT "DB_Outputs".cylinderDirectionB[6] AND NOT "DB_Outputs".vent[6])));
   "DB_Outputs".cylinderDirectionAActive[6] := ("automaticMode" AND "DB_Outputs".active.%X12) OR ("manualMode" AND ("DB_Outputs".cylinderDirectionA[6] OR ("DB_Outputs".cylinderDirectionAActive[6] AND NOT "DB_Outputs".cylinderDirectionB[6] AND NOT "DB_Outputs".vent[6])));
   "qcylinder7DirectionA" := #_w1;
END_REGION

REGION Network 17: RET CYL 7.- SPARE
   RUNG wire#powerrail
      Contact( "automaticMode" )
      Contact( "DB_Outputs".active.%X13 )
      wire#w1
      Coil( "DB_Outputs".cylinderDirectionBActive[6] )
   END_RUNG
   RUNG wire#powerrail
      Contact( "manualMode" )
      wire#w2
      Contact( "DB_Outputs".cylinderDirectionB[6] )
   END_RUNG wire#w1
   RUNG wire#w2
      Contact( "DB_Outputs".cylinderDirectionBActive[6] )
      I_Contact( "DB_Outputs".cylinderDirectionA[6] )
      I_Contact( "DB_Outputs".vent[6] )
   END_RUNG wire#w1
   RUNG wire#w1
      Coil( "qcylinder7DirectionB" )
   END_RUNG
   // the same network as SCL:
   #_w1 := ("automaticMode" AND "DB_Outputs".active.%X13) OR ("manualMode" AND ("DB_Outputs".cylinderDirectionB[6] OR ("DB_Outputs".cylinderDirectionBActive[6] AND NOT "DB_Outputs".cylinderDirectionA[6] AND NOT "DB_Outputs".vent[6])));
   "DB_Outputs".cylinderDirectionBActive[6] := ("automaticMode" AND "DB_Outputs".active.%X13) OR ("manualMode" AND ("DB_Outputs".cylinderDirectionB[6] OR ("DB_Outputs".cylinderDirectionBActive[6] AND NOT "DB_Outputs".cylinderDirectionA[6] AND NOT "DB_Outputs".vent[6])));
   "qcylinder7DirectionB" := #_w1;
END_REGION

REGION Network 18: EXT CYL 8.- SPARE
   RUNG wire#powerrail
      Contact( "automaticMode" )
      Contact( "LOG0" )
      wire#w1
      Coil( "DB_Outputs".cylinderDirectionAActive[7] )
   END_RUNG
   RUNG wire#powerrail
      Contact( "manualMode" )
      wire#w2
      Contact( "DB_Outputs".cylinderDirectionA[7] )
   END_RUNG wire#w1
   RUNG wire#w2
      Contact( "DB_Outputs".cylinderDirectionAActive[7] )
      I_Contact( "DB_Outputs".cylinderDirectionB[7] )
      I_Contact( "DB_Outputs".vent[7] )
   END_RUNG wire#w1
   RUNG wire#w1
      Coil( "qcylinder8DirectionA" )
   END_RUNG
   // the same network as SCL:
   #_w1 := ("automaticMode" AND "LOG0") OR ("manualMode" AND ("DB_Outputs".cylinderDirectionA[7] OR ("DB_Outputs".cylinderDirectionAActive[7] AND NOT "DB_Outputs".cylinderDirectionB[7] AND NOT "DB_Outputs".vent[7])));
   "DB_Outputs".cylinderDirectionAActive[7] := ("automaticMode" AND "LOG0") OR ("manualMode" AND ("DB_Outputs".cylinderDirectionA[7] OR ("DB_Outputs".cylinderDirectionAActive[7] AND NOT "DB_Outputs".cylinderDirectionB[7] AND NOT "DB_Outputs".vent[7])));
   "qcylinder8DirectionA" := #_w1;
END_REGION

REGION Network 19: RET CYL 8.- SPARE
   RUNG wire#powerrail
      Contact( "automaticMode" )
      Contact( "LOG0" )
      wire#w1
      Coil( "DB_Outputs".cylinderDirectionBActive[7] )
   END_RUNG
   RUNG wire#powerrail
      Contact( "manualMode" )
      wire#w2
      Contact( "DB_Outputs".cylinderDirectionB[7] )
   END_RUNG wire#w1
   RUNG wire#w2
      Contact( "DB_Outputs".cylinderDirectionBActive[7] )
      I_Contact( "DB_Outputs".cylinderDirectionA[7] )
      I_Contact( "DB_Outputs".vent[7] )
   END_RUNG wire#w1
   RUNG wire#w1
      Coil( "qcylinder8DirectionB" )
   END_RUNG
   // the same network as SCL:
   #_w1 := ("automaticMode" AND "LOG0") OR ("manualMode" AND ("DB_Outputs".cylinderDirectionB[7] OR ("DB_Outputs".cylinderDirectionBActive[7] AND NOT "DB_Outputs".cylinderDirectionA[7] AND NOT "DB_Outputs".vent[7])));
   "DB_Outputs".cylinderDirectionBActive[7] := ("automaticMode" AND "LOG0") OR ("manualMode" AND ("DB_Outputs".cylinderDirectionB[7] OR ("DB_Outputs".cylinderDirectionBActive[7] AND NOT "DB_Outputs".cylinderDirectionA[7] AND NOT "DB_Outputs".vent[7])));
   "qcylinder8DirectionB" := #_w1;
END_REGION

REGION Network 20: EXT CYL 9.- SPARE
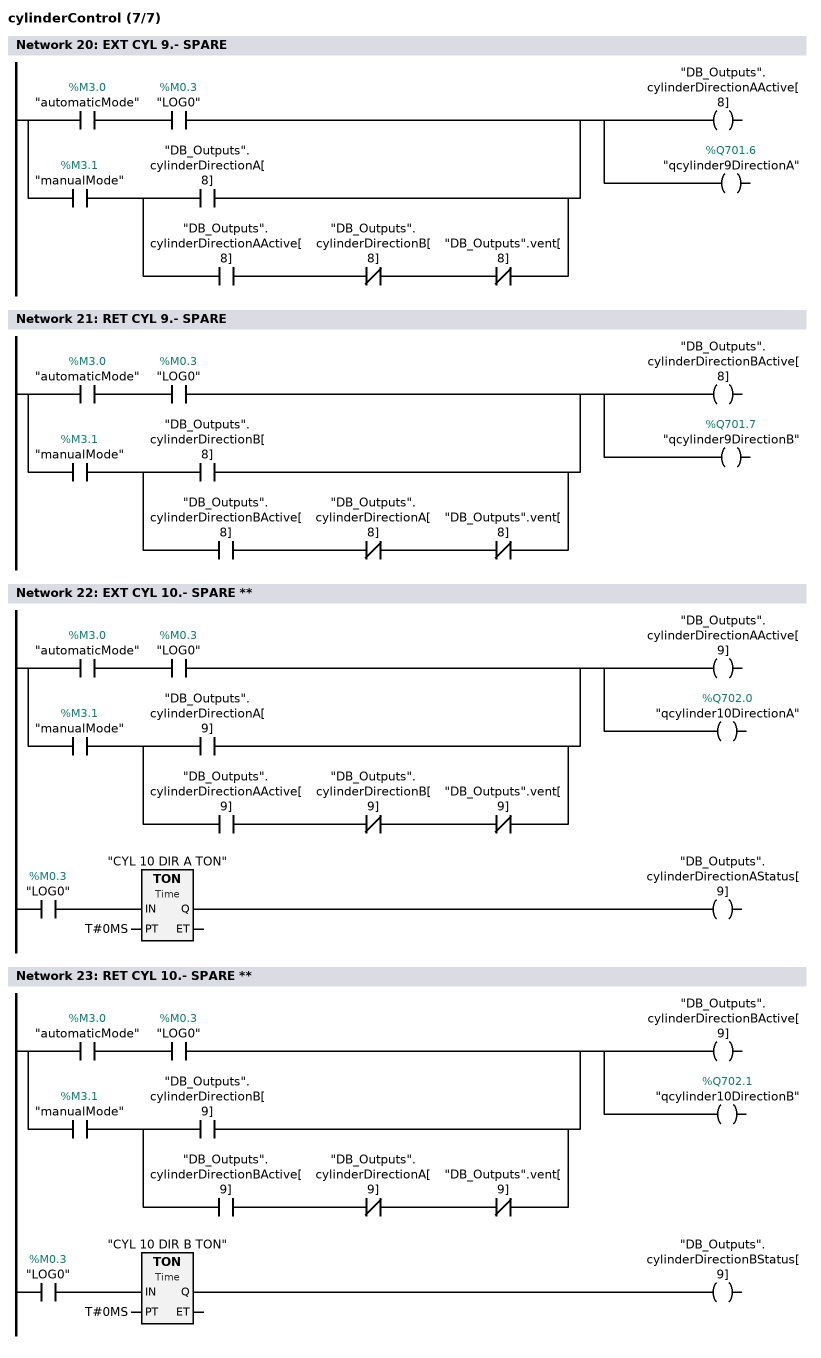
   RUNG wire#powerrail
      Contact( "automaticMode" )
      Contact( "LOG0" )
      wire#w1
      Coil( "DB_Outputs".cylinderDirectionAActive[8] )
   END_RUNG
   RUNG wire#powerrail
      Contact( "manualMode" )
      wire#w2
      Contact( "DB_Outputs".cylinderDirectionA[8] )
   END_RUNG wire#w1
   RUNG wire#w2
      Contact( "DB_Outputs".cylinderDirectionAActive[8] )
      I_Contact( "DB_Outputs".cylinderDirectionB[8] )
      I_Contact( "DB_Outputs".vent[8] )
   END_RUNG wire#w1
   RUNG wire#w1
      Coil( "qcylinder9DirectionA" )
   END_RUNG
   // the same network as SCL:
   #_w1 := ("automaticMode" AND "LOG0") OR ("manualMode" AND ("DB_Outputs".cylinderDirectionA[8] OR ("DB_Outputs".cylinderDirectionAActive[8] AND NOT "DB_Outputs".cylinderDirectionB[8] AND NOT "DB_Outputs".vent[8])));
   "DB_Outputs".cylinderDirectionAActive[8] := ("automaticMode" AND "LOG0") OR ("manualMode" AND ("DB_Outputs".cylinderDirectionA[8] OR ("DB_Outputs".cylinderDirectionAActive[8] AND NOT "DB_Outputs".cylinderDirectionB[8] AND NOT "DB_Outputs".vent[8])));
   "qcylinder9DirectionA" := #_w1;
END_REGION

REGION Network 21: RET CYL 9.- SPARE
   RUNG wire#powerrail
      Contact( "automaticMode" )
      Contact( "LOG0" )
      wire#w1
      Coil( "DB_Outputs".cylinderDirectionBActive[8] )
   END_RUNG
   RUNG wire#powerrail
      Contact( "manualMode" )
      wire#w2
      Contact( "DB_Outputs".cylinderDirectionB[8] )
   END_RUNG wire#w1
   RUNG wire#w2
      Contact( "DB_Outputs".cylinderDirectionBActive[8] )
      I_Contact( "DB_Outputs".cylinderDirectionA[8] )
      I_Contact( "DB_Outputs".vent[8] )
   END_RUNG wire#w1
   RUNG wire#w1
      Coil( "qcylinder9DirectionB" )
   END_RUNG
   // the same network as SCL:
   #_w1 := ("automaticMode" AND "LOG0") OR ("manualMode" AND ("DB_Outputs".cylinderDirectionB[8] OR ("DB_Outputs".cylinderDirectionBActive[8] AND NOT "DB_Outputs".cylinderDirectionA[8] AND NOT "DB_Outputs".vent[8])));
   "DB_Outputs".cylinderDirectionBActive[8] := ("automaticMode" AND "LOG0") OR ("manualMode" AND ("DB_Outputs".cylinderDirectionB[8] OR ("DB_Outputs".cylinderDirectionBActive[8] AND NOT "DB_Outputs".cylinderDirectionA[8] AND NOT "DB_Outputs".vent[8])));
   "qcylinder9DirectionB" := #_w1;
END_REGION

REGION Network 22: EXT CYL 10.- SPARE **
   RUNG wire#powerrail
      Contact( "automaticMode" )
      Contact( "LOG0" )
      wire#w1
      Coil( "DB_Outputs".cylinderDirectionAActive[9] )
   END_RUNG
   RUNG wire#powerrail
      Contact( "manualMode" )
      wire#w2
      Contact( "DB_Outputs".cylinderDirectionA[9] )
   END_RUNG wire#w1
   RUNG wire#w2
      Contact( "DB_Outputs".cylinderDirectionAActive[9] )
      I_Contact( "DB_Outputs".cylinderDirectionB[9] )
      I_Contact( "DB_Outputs".vent[9] )
   END_RUNG wire#w1
   RUNG wire#w1
      Coil( "qcylinder10DirectionA" )
   END_RUNG
   RUNG wire#powerrail
      Contact( "LOG0" )
      { S7_Templates := "time_type := Time" } "CYL 10 DIR A TON".TON(pt := T#0MS, et =>)
      Coil( "DB_Outputs".cylinderDirectionAStatus[9] )
   END_RUNG
   // the same network as SCL:
   #_w1 := ("automaticMode" AND "LOG0") OR ("manualMode" AND ("DB_Outputs".cylinderDirectionA[9] OR ("DB_Outputs".cylinderDirectionAActive[9] AND NOT "DB_Outputs".cylinderDirectionB[9] AND NOT "DB_Outputs".vent[9])));
   "DB_Outputs".cylinderDirectionAActive[9] := ("automaticMode" AND "LOG0") OR ("manualMode" AND ("DB_Outputs".cylinderDirectionA[9] OR ("DB_Outputs".cylinderDirectionAActive[9] AND NOT "DB_Outputs".cylinderDirectionB[9] AND NOT "DB_Outputs".vent[9])));
   "qcylinder10DirectionA" := #_w1;
   "CYL 10 DIR A TON".TON(IN := "LOG0", PT := T#0MS);
   "DB_Outputs".cylinderDirectionAStatus[9] := "CYL 10 DIR A TON".Q;
END_REGION

REGION Network 23: RET CYL 10.- SPARE **
   RUNG wire#powerrail
      Contact( "automaticMode" )
      Contact( "LOG0" )
      wire#w1
      Coil( "DB_Outputs".cylinderDirectionBActive[9] )
   END_RUNG
   RUNG wire#powerrail
      Contact( "manualMode" )
      wire#w2
      Contact( "DB_Outputs".cylinderDirectionB[9] )
   END_RUNG wire#w1
   RUNG wire#w2
      Contact( "DB_Outputs".cylinderDirectionBActive[9] )
      I_Contact( "DB_Outputs".cylinderDirectionA[9] )
      I_Contact( "DB_Outputs".vent[9] )
   END_RUNG wire#w1
   RUNG wire#w1
      Coil( "qcylinder10DirectionB" )
   END_RUNG
   RUNG wire#powerrail
      Contact( "LOG0" )
      { S7_Templates := "time_type := Time" } "CYL 10 DIR B TON".TON(pt := T#0MS, et =>)
      Coil( "DB_Outputs".cylinderDirectionBStatus[9] )
   END_RUNG
   // the same network as SCL:
   #_w1 := ("automaticMode" AND "LOG0") OR ("manualMode" AND ("DB_Outputs".cylinderDirectionB[9] OR ("DB_Outputs".cylinderDirectionBActive[9] AND NOT "DB_Outputs".cylinderDirectionA[9] AND NOT "DB_Outputs".vent[9])));
   "DB_Outputs".cylinderDirectionBActive[9] := ("automaticMode" AND "LOG0") OR ("manualMode" AND ("DB_Outputs".cylinderDirectionB[9] OR ("DB_Outputs".cylinderDirectionBActive[9] AND NOT "DB_Outputs".cylinderDirectionA[9] AND NOT "DB_Outputs".vent[9])));
   "qcylinder10DirectionB" := #_w1;
   "CYL 10 DIR B TON".TON(IN := "LOG0", PT := T#0MS);
   "DB_Outputs".cylinderDirectionBStatus[9] := "CYL 10 DIR B TON".Q;
END_REGION
END_FUNCTION

FUNCTION "outputsMapping" : Void   // FC8, LAD
{ S7_Optimized_Access := 'TRUE' }
VERSION : 0.1
// stored: AutoNumber true, IsIECCheckEnabled false, SetENOAutomatically false, UDAEnableTagReadback false
BEGIN

REGION Network 1: OUTPUT VALVE ACTIVATION
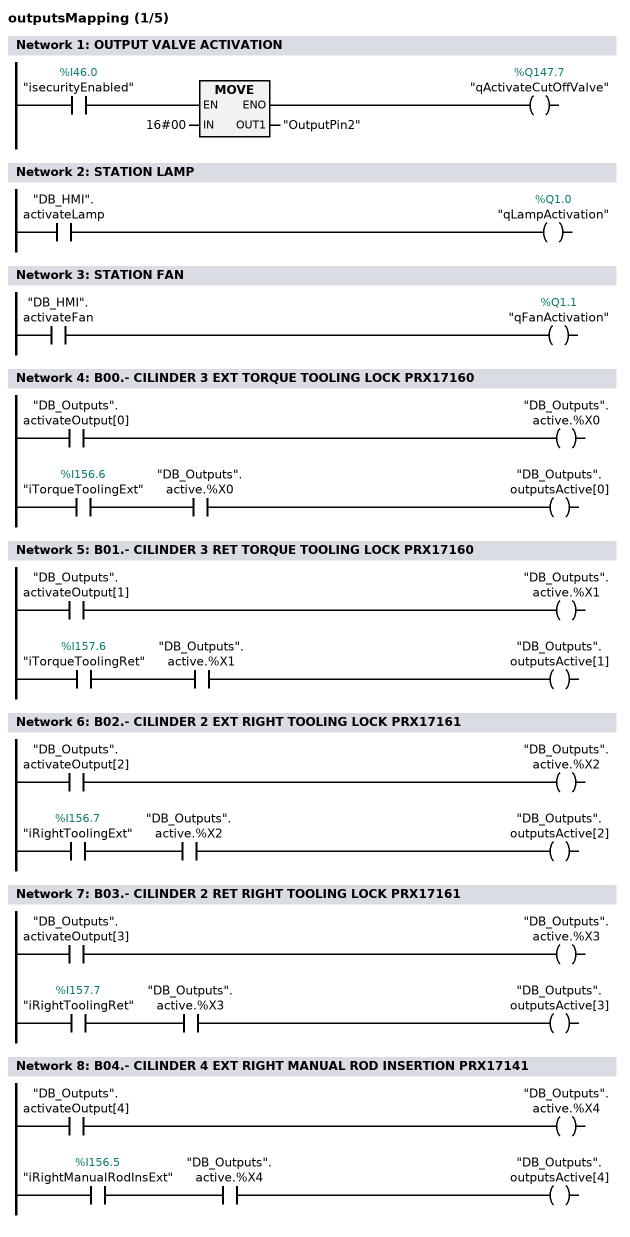
   RUNG wire#powerrail
      Contact( "isecurityEnabled" )
      Move(in := 16#00, out1 => "OutputPin2")
      Coil( "qActivateCutOffValve" )
   END_RUNG
   // the same network as SCL:
   IF "isecurityEnabled" THEN "OutputPin2" := 16#00; END_IF;
   "qActivateCutOffValve" := "isecurityEnabled";
END_REGION

REGION Network 2: STATION LAMP
   RUNG wire#powerrail
      Contact( "DB_HMI".activateLamp )
      Coil( "qLampActivation" )
   END_RUNG
   // the same network as SCL:
   "qLampActivation" := "DB_HMI".activateLamp;
END_REGION

REGION Network 3: STATION FAN
   RUNG wire#powerrail
      Contact( "DB_HMI".activateFan )
      Coil( "qFanActivation" )
   END_RUNG
   // the same network as SCL:
   "qFanActivation" := "DB_HMI".activateFan;
END_REGION

REGION Network 4: B00.- CILINDER 3 EXT TORQUE TOOLING LOCK PRX17160
   RUNG wire#powerrail
      Contact( "DB_Outputs".activateOutput[0] )
      Coil( "DB_Outputs".active.%X0 )
   END_RUNG
   RUNG wire#powerrail
      Contact( "iTorqueToolingExt" )
      Contact( "DB_Outputs".active.%X0 )
      Coil( "DB_Outputs".outputsActive[0] )
   END_RUNG
   // the same network as SCL:
   "DB_Outputs".active.%X0 := "DB_Outputs".activateOutput[0];
   "DB_Outputs".outputsActive[0] := "iTorqueToolingExt" AND "DB_Outputs".active.%X0;
END_REGION

REGION Network 5: B01.- CILINDER 3 RET TORQUE TOOLING LOCK PRX17160
   RUNG wire#powerrail
      Contact( "DB_Outputs".activateOutput[1] )
      Coil( "DB_Outputs".active.%X1 )
   END_RUNG
   RUNG wire#powerrail
      Contact( "iTorqueToolingRet" )
      Contact( "DB_Outputs".active.%X1 )
      Coil( "DB_Outputs".outputsActive[1] )
   END_RUNG
   // the same network as SCL:
   "DB_Outputs".active.%X1 := "DB_Outputs".activateOutput[1];
   "DB_Outputs".outputsActive[1] := "iTorqueToolingRet" AND "DB_Outputs".active.%X1;
END_REGION

REGION Network 6: B02.- CILINDER 2 EXT RIGHT TOOLING LOCK PRX17161
   RUNG wire#powerrail
      Contact( "DB_Outputs".activateOutput[2] )
      Coil( "DB_Outputs".active.%X2 )
   END_RUNG
   RUNG wire#powerrail
      Contact( "iRightToolingExt" )
      Contact( "DB_Outputs".active.%X2 )
      Coil( "DB_Outputs".outputsActive[2] )
   END_RUNG
   // the same network as SCL:
   "DB_Outputs".active.%X2 := "DB_Outputs".activateOutput[2];
   "DB_Outputs".outputsActive[2] := "iRightToolingExt" AND "DB_Outputs".active.%X2;
END_REGION

REGION Network 7: B03.- CILINDER 2 RET RIGHT TOOLING LOCK PRX17161
   RUNG wire#powerrail
      Contact( "DB_Outputs".activateOutput[3] )
      Coil( "DB_Outputs".active.%X3 )
   END_RUNG
   RUNG wire#powerrail
      Contact( "iRightToolingRet" )
      Contact( "DB_Outputs".active.%X3 )
      Coil( "DB_Outputs".outputsActive[3] )
   END_RUNG
   // the same network as SCL:
   "DB_Outputs".active.%X3 := "DB_Outputs".activateOutput[3];
   "DB_Outputs".outputsActive[3] := "iRightToolingRet" AND "DB_Outputs".active.%X3;
END_REGION

REGION Network 8: B04.- CILINDER 4 EXT RIGHT MANUAL ROD INSERTION PRX17141
   RUNG wire#powerrail
      Contact( "DB_Outputs".activateOutput[4] )
      Coil( "DB_Outputs".active.%X4 )
   END_RUNG
   RUNG wire#powerrail
      Contact( "iRightManualRodInsExt" )
      Contact( "DB_Outputs".active.%X4 )
      Coil( "DB_Outputs".outputsActive[4] )
   END_RUNG
   // the same network as SCL:
   "DB_Outputs".active.%X4 := "DB_Outputs".activateOutput[4];
   "DB_Outputs".outputsActive[4] := "iRightManualRodInsExt" AND "DB_Outputs".active.%X4;
END_REGION

REGION Network 9: B05.- CILINDER 4 RET RIGHT MANUAL ROD INSERTION PRX17141
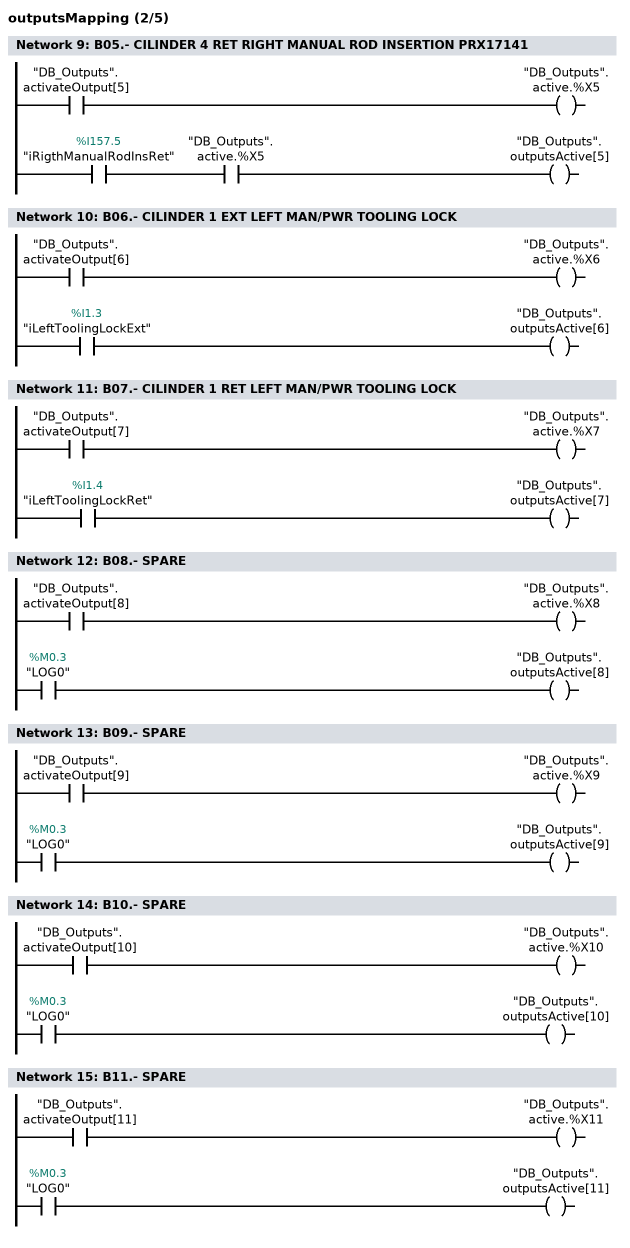
   RUNG wire#powerrail
      Contact( "DB_Outputs".activateOutput[5] )
      Coil( "DB_Outputs".active.%X5 )
   END_RUNG
   RUNG wire#powerrail
      Contact( "iRigthManualRodInsRet" )
      Contact( "DB_Outputs".active.%X5 )
      Coil( "DB_Outputs".outputsActive[5] )
   END_RUNG
   // the same network as SCL:
   "DB_Outputs".active.%X5 := "DB_Outputs".activateOutput[5];
   "DB_Outputs".outputsActive[5] := "iRigthManualRodInsRet" AND "DB_Outputs".active.%X5;
END_REGION

REGION Network 10: B06.- CILINDER 1 EXT LEFT MAN/PWR TOOLING LOCK
   RUNG wire#powerrail
      Contact( "DB_Outputs".activateOutput[6] )
      Coil( "DB_Outputs".active.%X6 )
   END_RUNG
   RUNG wire#powerrail
      Contact( "iLeftToolingLockExt" )
      Coil( "DB_Outputs".outputsActive[6] )
   END_RUNG
   // the same network as SCL:
   "DB_Outputs".active.%X6 := "DB_Outputs".activateOutput[6];
   "DB_Outputs".outputsActive[6] := "iLeftToolingLockExt";
END_REGION

REGION Network 11: B07.- CILINDER 1 RET LEFT MAN/PWR TOOLING LOCK
   RUNG wire#powerrail
      Contact( "DB_Outputs".activateOutput[7] )
      Coil( "DB_Outputs".active.%X7 )
   END_RUNG
   RUNG wire#powerrail
      Contact( "iLeftToolingLockRet" )
      Coil( "DB_Outputs".outputsActive[7] )
   END_RUNG
   // the same network as SCL:
   "DB_Outputs".active.%X7 := "DB_Outputs".activateOutput[7];
   "DB_Outputs".outputsActive[7] := "iLeftToolingLockRet";
END_REGION

REGION Network 12: B08.- SPARE
   RUNG wire#powerrail
      Contact( "DB_Outputs".activateOutput[8] )
      Coil( "DB_Outputs".active.%X8 )
   END_RUNG
   RUNG wire#powerrail
      Contact( "LOG0" )
      Coil( "DB_Outputs".outputsActive[8] )
   END_RUNG
   // the same network as SCL:
   "DB_Outputs".active.%X8 := "DB_Outputs".activateOutput[8];
   "DB_Outputs".outputsActive[8] := "LOG0";
END_REGION

REGION Network 13: B09.- SPARE
   RUNG wire#powerrail
      Contact( "DB_Outputs".activateOutput[9] )
      Coil( "DB_Outputs".active.%X9 )
   END_RUNG
   RUNG wire#powerrail
      Contact( "LOG0" )
      Coil( "DB_Outputs".outputsActive[9] )
   END_RUNG
   // the same network as SCL:
   "DB_Outputs".active.%X9 := "DB_Outputs".activateOutput[9];
   "DB_Outputs".outputsActive[9] := "LOG0";
END_REGION

REGION Network 14: B10.- SPARE
   RUNG wire#powerrail
      Contact( "DB_Outputs".activateOutput[10] )
      Coil( "DB_Outputs".active.%X10 )
   END_RUNG
   RUNG wire#powerrail
      Contact( "LOG0" )
      Coil( "DB_Outputs".outputsActive[10] )
   END_RUNG
   // the same network as SCL:
   "DB_Outputs".active.%X10 := "DB_Outputs".activateOutput[10];
   "DB_Outputs".outputsActive[10] := "LOG0";
END_REGION

REGION Network 15: B11.- SPARE
   RUNG wire#powerrail
      Contact( "DB_Outputs".activateOutput[11] )
      Coil( "DB_Outputs".active.%X11 )
   END_RUNG
   RUNG wire#powerrail
      Contact( "LOG0" )
      Coil( "DB_Outputs".outputsActive[11] )
   END_RUNG
   // the same network as SCL:
   "DB_Outputs".active.%X11 := "DB_Outputs".activateOutput[11];
   "DB_Outputs".outputsActive[11] := "LOG0";
END_REGION

REGION Network 16: B12.- CILINDER 7 EXT INSERTION CYLINDERS WASHER/ROD
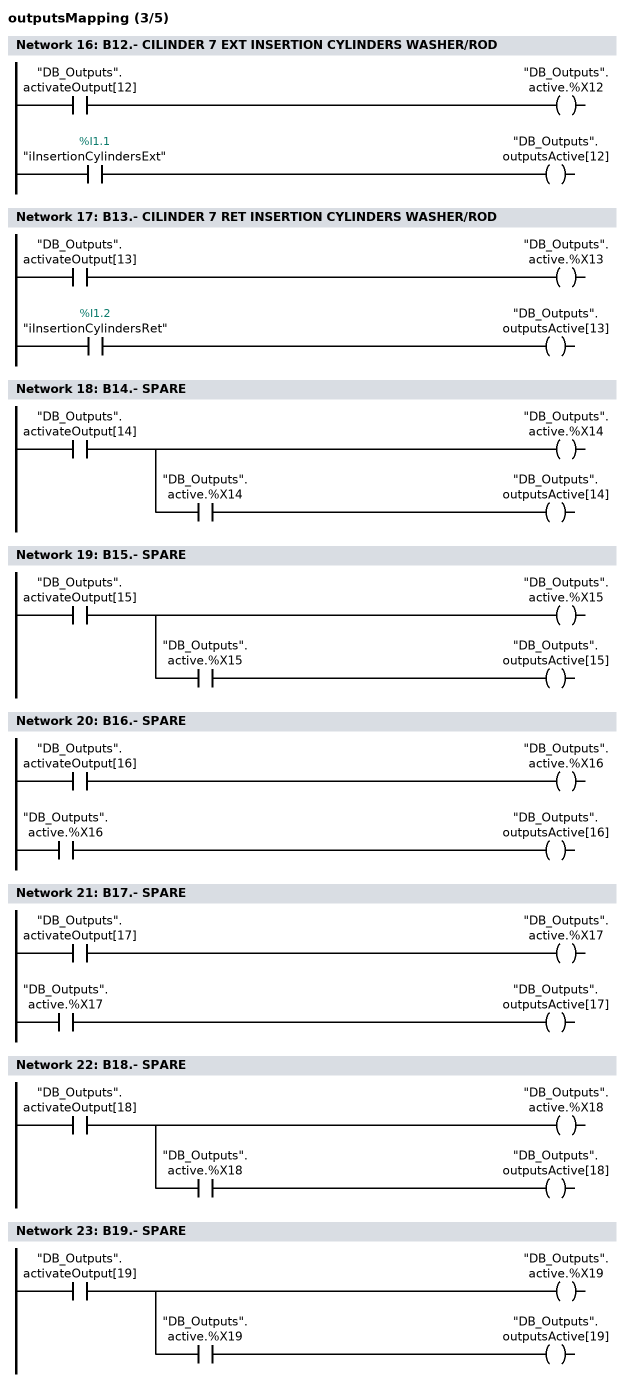
   RUNG wire#powerrail
      Contact( "DB_Outputs".activateOutput[12] )
      Coil( "DB_Outputs".active.%X12 )
   END_RUNG
   RUNG wire#powerrail
      Contact( "iInsertionCylindersExt" )
      Coil( "DB_Outputs".outputsActive[12] )
   END_RUNG
   // the same network as SCL:
   "DB_Outputs".active.%X12 := "DB_Outputs".activateOutput[12];
   "DB_Outputs".outputsActive[12] := "iInsertionCylindersExt";
END_REGION

REGION Network 17: B13.- CILINDER 7 RET INSERTION CYLINDERS WASHER/ROD
   RUNG wire#powerrail
      Contact( "DB_Outputs".activateOutput[13] )
      Coil( "DB_Outputs".active.%X13 )
   END_RUNG
   RUNG wire#powerrail
      Contact( "iInsertionCylindersRet" )
      Coil( "DB_Outputs".outputsActive[13] )
   END_RUNG
   // the same network as SCL:
   "DB_Outputs".active.%X13 := "DB_Outputs".activateOutput[13];
   "DB_Outputs".outputsActive[13] := "iInsertionCylindersRet";
END_REGION

REGION Network 18: B14.- SPARE
   RUNG wire#powerrail
      Contact( "DB_Outputs".activateOutput[14] )
      wire#w1
      Coil( "DB_Outputs".active.%X14 )
   END_RUNG
   RUNG wire#w1
      Contact( "DB_Outputs".active.%X14 )
      Coil( "DB_Outputs".outputsActive[14] )
   END_RUNG
   // the same network as SCL:
   "DB_Outputs".active.%X14 := "DB_Outputs".activateOutput[14];
   "DB_Outputs".outputsActive[14] := "DB_Outputs".activateOutput[14] AND "DB_Outputs".active.%X14;
END_REGION

REGION Network 19: B15.- SPARE
   RUNG wire#powerrail
      Contact( "DB_Outputs".activateOutput[15] )
      wire#w1
      Coil( "DB_Outputs".active.%X15 )
   END_RUNG
   RUNG wire#w1
      Contact( "DB_Outputs".active.%X15 )
      Coil( "DB_Outputs".outputsActive[15] )
   END_RUNG
   // the same network as SCL:
   "DB_Outputs".active.%X15 := "DB_Outputs".activateOutput[15];
   "DB_Outputs".outputsActive[15] := "DB_Outputs".activateOutput[15] AND "DB_Outputs".active.%X15;
END_REGION

REGION Network 20: B16.- SPARE
   RUNG wire#powerrail
      Contact( "DB_Outputs".activateOutput[16] )
      Coil( "DB_Outputs".active.%X16 )
   END_RUNG
   RUNG wire#powerrail
      Contact( "DB_Outputs".active.%X16 )
      Coil( "DB_Outputs".outputsActive[16] )
   END_RUNG
   // the same network as SCL:
   "DB_Outputs".active.%X16 := "DB_Outputs".activateOutput[16];
   "DB_Outputs".outputsActive[16] := "DB_Outputs".active.%X16;
END_REGION

REGION Network 21: B17.- SPARE
   RUNG wire#powerrail
      Contact( "DB_Outputs".activateOutput[17] )
      Coil( "DB_Outputs".active.%X17 )
   END_RUNG
   RUNG wire#powerrail
      Contact( "DB_Outputs".active.%X17 )
      Coil( "DB_Outputs".outputsActive[17] )
   END_RUNG
   // the same network as SCL:
   "DB_Outputs".active.%X17 := "DB_Outputs".activateOutput[17];
   "DB_Outputs".outputsActive[17] := "DB_Outputs".active.%X17;
END_REGION

REGION Network 22: B18.- SPARE
   RUNG wire#powerrail
      Contact( "DB_Outputs".activateOutput[18] )
      wire#w1
      Coil( "DB_Outputs".active.%X18 )
   END_RUNG
   RUNG wire#w1
      Contact( "DB_Outputs".active.%X18 )
      Coil( "DB_Outputs".outputsActive[18] )
   END_RUNG
   // the same network as SCL:
   "DB_Outputs".active.%X18 := "DB_Outputs".activateOutput[18];
   "DB_Outputs".outputsActive[18] := "DB_Outputs".activateOutput[18] AND "DB_Outputs".active.%X18;
END_REGION

REGION Network 23: B19.- SPARE
   RUNG wire#powerrail
      Contact( "DB_Outputs".activateOutput[19] )
      wire#w1
      Coil( "DB_Outputs".active.%X19 )
   END_RUNG
   RUNG wire#w1
      Contact( "DB_Outputs".active.%X19 )
      Coil( "DB_Outputs".outputsActive[19] )
   END_RUNG
   // the same network as SCL:
   "DB_Outputs".active.%X19 := "DB_Outputs".activateOutput[19];
   "DB_Outputs".outputsActive[19] := "DB_Outputs".activateOutput[19] AND "DB_Outputs".active.%X19;
END_REGION

REGION Network 24: B20.- SPARE
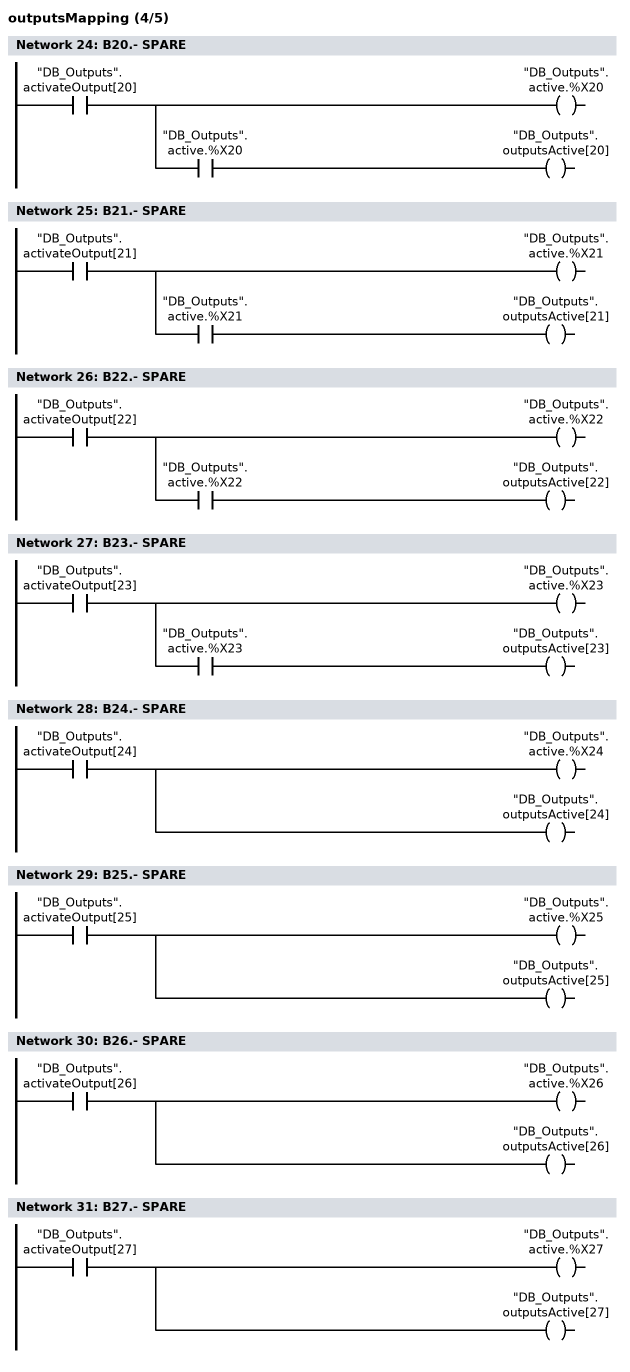
   RUNG wire#powerrail
      Contact( "DB_Outputs".activateOutput[20] )
      wire#w1
      Coil( "DB_Outputs".active.%X20 )
   END_RUNG
   RUNG wire#w1
      Contact( "DB_Outputs".active.%X20 )
      Coil( "DB_Outputs".outputsActive[20] )
   END_RUNG
   // the same network as SCL:
   "DB_Outputs".active.%X20 := "DB_Outputs".activateOutput[20];
   "DB_Outputs".outputsActive[20] := "DB_Outputs".activateOutput[20] AND "DB_Outputs".active.%X20;
END_REGION

REGION Network 25: B21.- SPARE
   RUNG wire#powerrail
      Contact( "DB_Outputs".activateOutput[21] )
      wire#w1
      Coil( "DB_Outputs".active.%X21 )
   END_RUNG
   RUNG wire#w1
      Contact( "DB_Outputs".active.%X21 )
      Coil( "DB_Outputs".outputsActive[21] )
   END_RUNG
   // the same network as SCL:
   "DB_Outputs".active.%X21 := "DB_Outputs".activateOutput[21];
   "DB_Outputs".outputsActive[21] := "DB_Outputs".activateOutput[21] AND "DB_Outputs".active.%X21;
END_REGION

REGION Network 26: B22.- SPARE
   RUNG wire#powerrail
      Contact( "DB_Outputs".activateOutput[22] )
      wire#w1
      Coil( "DB_Outputs".active.%X22 )
   END_RUNG
   RUNG wire#w1
      Contact( "DB_Outputs".active.%X22 )
      Coil( "DB_Outputs".outputsActive[22] )
   END_RUNG
   // the same network as SCL:
   "DB_Outputs".active.%X22 := "DB_Outputs".activateOutput[22];
   "DB_Outputs".outputsActive[22] := "DB_Outputs".activateOutput[22] AND "DB_Outputs".active.%X22;
END_REGION

REGION Network 27: B23.- SPARE
   RUNG wire#powerrail
      Contact( "DB_Outputs".activateOutput[23] )
      wire#w1
      Coil( "DB_Outputs".active.%X23 )
   END_RUNG
   RUNG wire#w1
      Contact( "DB_Outputs".active.%X23 )
      Coil( "DB_Outputs".outputsActive[23] )
   END_RUNG
   // the same network as SCL:
   "DB_Outputs".active.%X23 := "DB_Outputs".activateOutput[23];
   "DB_Outputs".outputsActive[23] := "DB_Outputs".activateOutput[23] AND "DB_Outputs".active.%X23;
END_REGION

REGION Network 28: B24.- SPARE
   RUNG wire#powerrail
      Contact( "DB_Outputs".activateOutput[24] )
      wire#w1
      Coil( "DB_Outputs".active.%X24 )
   END_RUNG
   RUNG wire#w1
      Coil( "DB_Outputs".outputsActive[24] )
   END_RUNG
   // the same network as SCL:
   "DB_Outputs".active.%X24 := "DB_Outputs".activateOutput[24];
   "DB_Outputs".outputsActive[24] := "DB_Outputs".activateOutput[24];
END_REGION

REGION Network 29: B25.- SPARE
   RUNG wire#powerrail
      Contact( "DB_Outputs".activateOutput[25] )
      wire#w1
      Coil( "DB_Outputs".active.%X25 )
   END_RUNG
   RUNG wire#w1
      Coil( "DB_Outputs".outputsActive[25] )
   END_RUNG
   // the same network as SCL:
   "DB_Outputs".active.%X25 := "DB_Outputs".activateOutput[25];
   "DB_Outputs".outputsActive[25] := "DB_Outputs".activateOutput[25];
END_REGION

REGION Network 30: B26.- SPARE
   RUNG wire#powerrail
      Contact( "DB_Outputs".activateOutput[26] )
      wire#w1
      Coil( "DB_Outputs".active.%X26 )
   END_RUNG
   RUNG wire#w1
      Coil( "DB_Outputs".outputsActive[26] )
   END_RUNG
   // the same network as SCL:
   "DB_Outputs".active.%X26 := "DB_Outputs".activateOutput[26];
   "DB_Outputs".outputsActive[26] := "DB_Outputs".activateOutput[26];
END_REGION

REGION Network 31: B27.- SPARE
   RUNG wire#powerrail
      Contact( "DB_Outputs".activateOutput[27] )
      wire#w1
      Coil( "DB_Outputs".active.%X27 )
   END_RUNG
   RUNG wire#w1
      Coil( "DB_Outputs".outputsActive[27] )
   END_RUNG
   // the same network as SCL:
   "DB_Outputs".active.%X27 := "DB_Outputs".activateOutput[27];
   "DB_Outputs".outputsActive[27] := "DB_Outputs".activateOutput[27];
END_REGION

REGION Network 32: B28.- SPARE
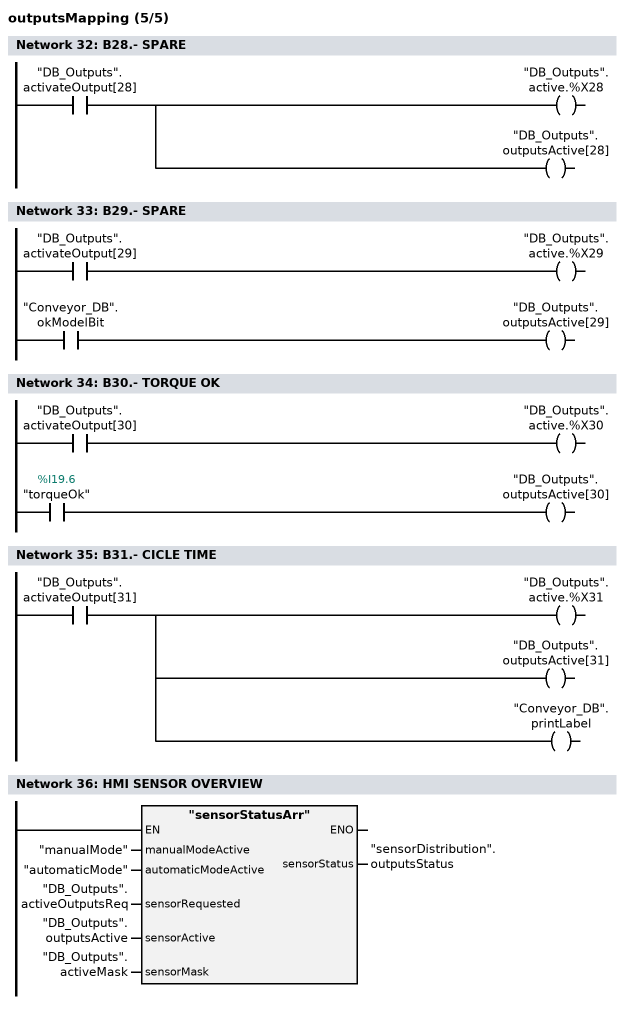
   RUNG wire#powerrail
      Contact( "DB_Outputs".activateOutput[28] )
      wire#w1
      Coil( "DB_Outputs".active.%X28 )
   END_RUNG
   RUNG wire#w1
      Coil( "DB_Outputs".outputsActive[28] )
   END_RUNG
   // the same network as SCL:
   "DB_Outputs".active.%X28 := "DB_Outputs".activateOutput[28];
   "DB_Outputs".outputsActive[28] := "DB_Outputs".activateOutput[28];
END_REGION

REGION Network 33: B29.- SPARE
   RUNG wire#powerrail
      Contact( "DB_Outputs".activateOutput[29] )
      Coil( "DB_Outputs".active.%X29 )
   END_RUNG
   RUNG wire#powerrail
      Contact( "Conveyor_DB".okModelBit )
      Coil( "DB_Outputs".outputsActive[29] )
   END_RUNG
   // the same network as SCL:
   "DB_Outputs".active.%X29 := "DB_Outputs".activateOutput[29];
   "DB_Outputs".outputsActive[29] := "Conveyor_DB".okModelBit;
END_REGION

REGION Network 34: B30.- TORQUE OK
   RUNG wire#powerrail
      Contact( "DB_Outputs".activateOutput[30] )
      Coil( "DB_Outputs".active.%X30 )
   END_RUNG
   RUNG wire#powerrail
      Contact( "torqueOk" )
      Coil( "DB_Outputs".outputsActive[30] )
   END_RUNG
   // the same network as SCL:
   "DB_Outputs".active.%X30 := "DB_Outputs".activateOutput[30];
   "DB_Outputs".outputsActive[30] := "torqueOk";
END_REGION

REGION Network 35: B31.- CICLE TIME
   RUNG wire#powerrail
      Contact( "DB_Outputs".activateOutput[31] )
      wire#w1
      Coil( "DB_Outputs".active.%X31 )
   END_RUNG
   RUNG wire#w1
      Coil( "DB_Outputs".outputsActive[31] )
   END_RUNG
   RUNG wire#w1
      Coil( "Conveyor_DB".printLabel )
   END_RUNG
   // the same network as SCL:
   "DB_Outputs".active.%X31 := "DB_Outputs".activateOutput[31];
   "DB_Outputs".outputsActive[31] := "DB_Outputs".activateOutput[31];
   "Conveyor_DB".printLabel := "DB_Outputs".activateOutput[31];
END_REGION

REGION Network 36: HMI SENSOR OVERVIEW
   RUNG wire#powerrail
      "sensorStatusArr"(manualModeActive := "manualMode", automaticModeActive := "automaticMode", sensorRequested := "DB_Outputs".activeOutputsReq, sensorActive := "DB_Outputs".outputsActive, sensorMask := "DB_Outputs".activeMask, sensorStatus => "sensorDistribution".outputsStatus)
   END_RUNG
   // the same network as SCL:
   "sensorStatusArr"(manualModeActive := "manualMode",
                     automaticModeActive := "automaticMode",
                     sensorRequested := "DB_Outputs".activeOutputsReq,
                     sensorActive := "DB_Outputs".outputsActive,
                     sensorMask := "DB_Outputs".activeMask,
                     sensorStatus => "sensorDistribution".outputsStatus);
END_REGION
END_FUNCTION

FUNCTION "sensorStatusArr" : Void   // FC38, LAD
{ S7_Optimized_Access := 'TRUE' }
VERSION : 0.1
// stored: AutoNumber true, IsIECCheckEnabled false, SetENOAutomatically false, UDAEnableTagReadback false
   VAR_INPUT
      manualModeActive : Bool;
      automaticModeActive : Bool;
      sensorRequested : Array[0..31] of Bool;
      sensorActive : Array[0..31] of Bool;
      sensorMask : Array[0..31] of Bool;
   END_VAR
   VAR_OUTPUT
      sensorStatus : Array[0..31] of Byte;
   END_VAR
BEGIN

REGION Network 1: Status 0
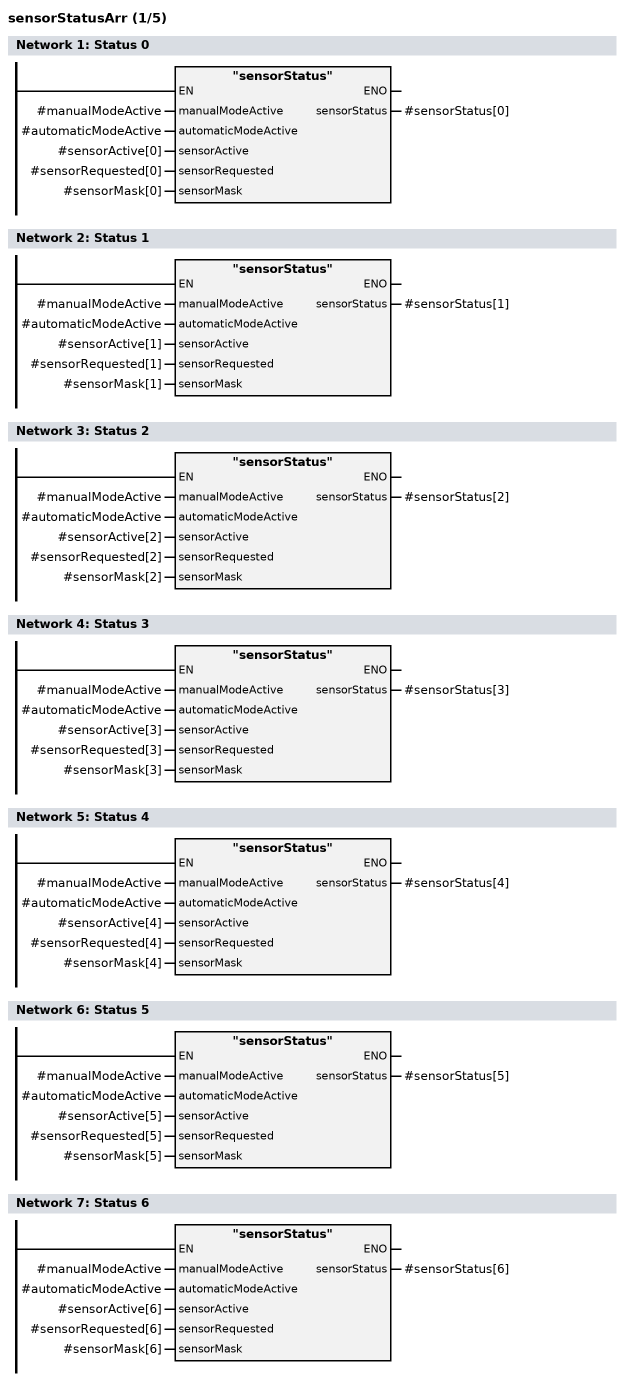
   RUNG wire#powerrail
      "sensorStatus"(manualModeActive := #manualModeActive, automaticModeActive := #automaticModeActive, sensorActive := #sensorActive[0], sensorRequested := #sensorRequested[0], sensorMask := #sensorMask[0], sensorStatus => #sensorStatus[0])
   END_RUNG
   // the same network as SCL:
   "sensorStatus"(manualModeActive := #manualModeActive,
                  automaticModeActive := #automaticModeActive,
                  sensorActive := #sensorActive[0],
                  sensorRequested := #sensorRequested[0],
                  sensorMask := #sensorMask[0],
                  sensorStatus => #sensorStatus[0]);
END_REGION

REGION Network 2: Status 1
   RUNG wire#powerrail
      "sensorStatus"(manualModeActive := #manualModeActive, automaticModeActive := #automaticModeActive, sensorActive := #sensorActive[1], sensorRequested := #sensorRequested[1], sensorMask := #sensorMask[1], sensorStatus => #sensorStatus[1])
   END_RUNG
   // the same network as SCL:
   "sensorStatus"(manualModeActive := #manualModeActive,
                  automaticModeActive := #automaticModeActive,
                  sensorActive := #sensorActive[1],
                  sensorRequested := #sensorRequested[1],
                  sensorMask := #sensorMask[1],
                  sensorStatus => #sensorStatus[1]);
END_REGION

REGION Network 3: Status 2
   RUNG wire#powerrail
      "sensorStatus"(manualModeActive := #manualModeActive, automaticModeActive := #automaticModeActive, sensorActive := #sensorActive[2], sensorRequested := #sensorRequested[2], sensorMask := #sensorMask[2], sensorStatus => #sensorStatus[2])
   END_RUNG
   // the same network as SCL:
   "sensorStatus"(manualModeActive := #manualModeActive,
                  automaticModeActive := #automaticModeActive,
                  sensorActive := #sensorActive[2],
                  sensorRequested := #sensorRequested[2],
                  sensorMask := #sensorMask[2],
                  sensorStatus => #sensorStatus[2]);
END_REGION

REGION Network 4: Status 3
   RUNG wire#powerrail
      "sensorStatus"(manualModeActive := #manualModeActive, automaticModeActive := #automaticModeActive, sensorActive := #sensorActive[3], sensorRequested := #sensorRequested[3], sensorMask := #sensorMask[3], sensorStatus => #sensorStatus[3])
   END_RUNG
   // the same network as SCL:
   "sensorStatus"(manualModeActive := #manualModeActive,
                  automaticModeActive := #automaticModeActive,
                  sensorActive := #sensorActive[3],
                  sensorRequested := #sensorRequested[3],
                  sensorMask := #sensorMask[3],
                  sensorStatus => #sensorStatus[3]);
END_REGION

REGION Network 5: Status 4
   RUNG wire#powerrail
      "sensorStatus"(manualModeActive := #manualModeActive, automaticModeActive := #automaticModeActive, sensorActive := #sensorActive[4], sensorRequested := #sensorRequested[4], sensorMask := #sensorMask[4], sensorStatus => #sensorStatus[4])
   END_RUNG
   // the same network as SCL:
   "sensorStatus"(manualModeActive := #manualModeActive,
                  automaticModeActive := #automaticModeActive,
                  sensorActive := #sensorActive[4],
                  sensorRequested := #sensorRequested[4],
                  sensorMask := #sensorMask[4],
                  sensorStatus => #sensorStatus[4]);
END_REGION

REGION Network 6: Status 5
   RUNG wire#powerrail
      "sensorStatus"(manualModeActive := #manualModeActive, automaticModeActive := #automaticModeActive, sensorActive := #sensorActive[5], sensorRequested := #sensorRequested[5], sensorMask := #sensorMask[5], sensorStatus => #sensorStatus[5])
   END_RUNG
   // the same network as SCL:
   "sensorStatus"(manualModeActive := #manualModeActive,
                  automaticModeActive := #automaticModeActive,
                  sensorActive := #sensorActive[5],
                  sensorRequested := #sensorRequested[5],
                  sensorMask := #sensorMask[5],
                  sensorStatus => #sensorStatus[5]);
END_REGION

REGION Network 7: Status 6
   RUNG wire#powerrail
      "sensorStatus"(manualModeActive := #manualModeActive, automaticModeActive := #automaticModeActive, sensorActive := #sensorActive[6], sensorRequested := #sensorRequested[6], sensorMask := #sensorMask[6], sensorStatus => #sensorStatus[6])
   END_RUNG
   // the same network as SCL:
   "sensorStatus"(manualModeActive := #manualModeActive,
                  automaticModeActive := #automaticModeActive,
                  sensorActive := #sensorActive[6],
                  sensorRequested := #sensorRequested[6],
                  sensorMask := #sensorMask[6],
                  sensorStatus => #sensorStatus[6]);
END_REGION

REGION Network 8: Status 7
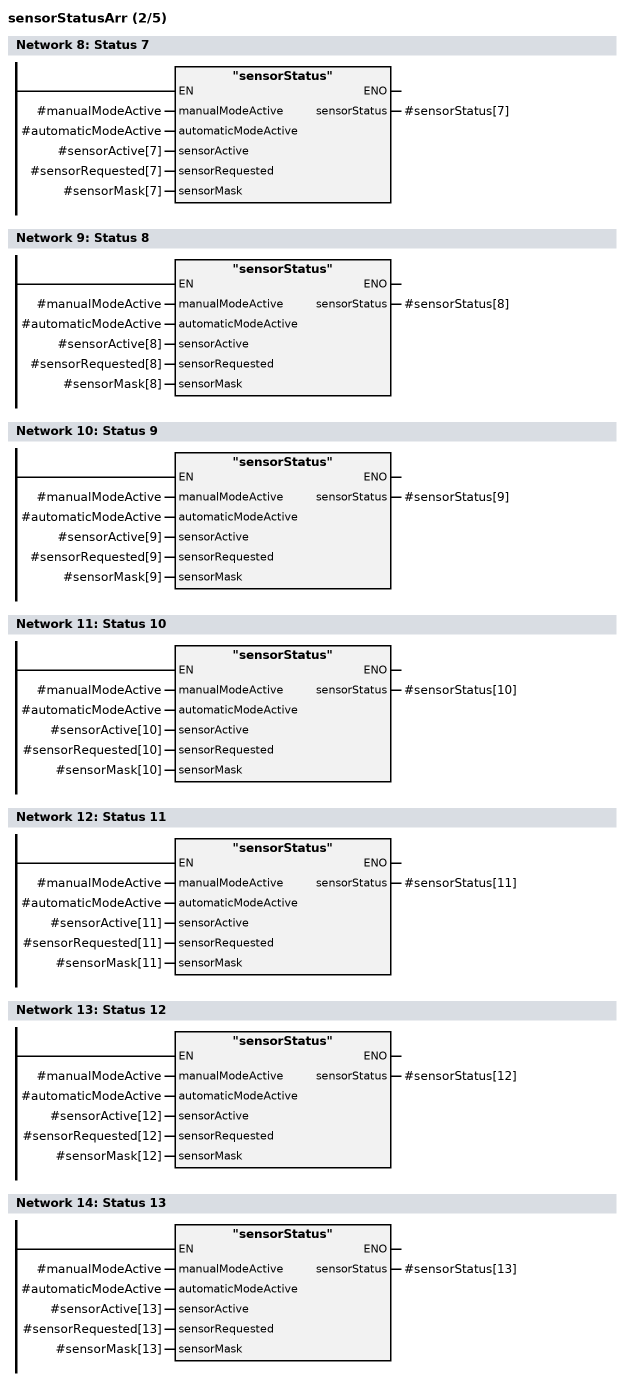
   RUNG wire#powerrail
      "sensorStatus"(manualModeActive := #manualModeActive, automaticModeActive := #automaticModeActive, sensorActive := #sensorActive[7], sensorRequested := #sensorRequested[7], sensorMask := #sensorMask[7], sensorStatus => #sensorStatus[7])
   END_RUNG
   // the same network as SCL:
   "sensorStatus"(manualModeActive := #manualModeActive,
                  automaticModeActive := #automaticModeActive,
                  sensorActive := #sensorActive[7],
                  sensorRequested := #sensorRequested[7],
                  sensorMask := #sensorMask[7],
                  sensorStatus => #sensorStatus[7]);
END_REGION

REGION Network 9: Status 8
   RUNG wire#powerrail
      "sensorStatus"(manualModeActive := #manualModeActive, automaticModeActive := #automaticModeActive, sensorActive := #sensorActive[8], sensorRequested := #sensorRequested[8], sensorMask := #sensorMask[8], sensorStatus => #sensorStatus[8])
   END_RUNG
   // the same network as SCL:
   "sensorStatus"(manualModeActive := #manualModeActive,
                  automaticModeActive := #automaticModeActive,
                  sensorActive := #sensorActive[8],
                  sensorRequested := #sensorRequested[8],
                  sensorMask := #sensorMask[8],
                  sensorStatus => #sensorStatus[8]);
END_REGION

REGION Network 10: Status 9
   RUNG wire#powerrail
      "sensorStatus"(manualModeActive := #manualModeActive, automaticModeActive := #automaticModeActive, sensorActive := #sensorActive[9], sensorRequested := #sensorRequested[9], sensorMask := #sensorMask[9], sensorStatus => #sensorStatus[9])
   END_RUNG
   // the same network as SCL:
   "sensorStatus"(manualModeActive := #manualModeActive,
                  automaticModeActive := #automaticModeActive,
                  sensorActive := #sensorActive[9],
                  sensorRequested := #sensorRequested[9],
                  sensorMask := #sensorMask[9],
                  sensorStatus => #sensorStatus[9]);
END_REGION

REGION Network 11: Status 10
   RUNG wire#powerrail
      "sensorStatus"(manualModeActive := #manualModeActive, automaticModeActive := #automaticModeActive, sensorActive := #sensorActive[10], sensorRequested := #sensorRequested[10], sensorMask := #sensorMask[10], sensorStatus => #sensorStatus[10])
   END_RUNG
   // the same network as SCL:
   "sensorStatus"(manualModeActive := #manualModeActive,
                  automaticModeActive := #automaticModeActive,
                  sensorActive := #sensorActive[10],
                  sensorRequested := #sensorRequested[10],
                  sensorMask := #sensorMask[10],
                  sensorStatus => #sensorStatus[10]);
END_REGION

REGION Network 12: Status 11
   RUNG wire#powerrail
      "sensorStatus"(manualModeActive := #manualModeActive, automaticModeActive := #automaticModeActive, sensorActive := #sensorActive[11], sensorRequested := #sensorRequested[11], sensorMask := #sensorMask[11], sensorStatus => #sensorStatus[11])
   END_RUNG
   // the same network as SCL:
   "sensorStatus"(manualModeActive := #manualModeActive,
                  automaticModeActive := #automaticModeActive,
                  sensorActive := #sensorActive[11],
                  sensorRequested := #sensorRequested[11],
                  sensorMask := #sensorMask[11],
                  sensorStatus => #sensorStatus[11]);
END_REGION

REGION Network 13: Status 12
   RUNG wire#powerrail
      "sensorStatus"(manualModeActive := #manualModeActive, automaticModeActive := #automaticModeActive, sensorActive := #sensorActive[12], sensorRequested := #sensorRequested[12], sensorMask := #sensorMask[12], sensorStatus => #sensorStatus[12])
   END_RUNG
   // the same network as SCL:
   "sensorStatus"(manualModeActive := #manualModeActive,
                  automaticModeActive := #automaticModeActive,
                  sensorActive := #sensorActive[12],
                  sensorRequested := #sensorRequested[12],
                  sensorMask := #sensorMask[12],
                  sensorStatus => #sensorStatus[12]);
END_REGION

REGION Network 14: Status 13
   RUNG wire#powerrail
      "sensorStatus"(manualModeActive := #manualModeActive, automaticModeActive := #automaticModeActive, sensorActive := #sensorActive[13], sensorRequested := #sensorRequested[13], sensorMask := #sensorMask[13], sensorStatus => #sensorStatus[13])
   END_RUNG
   // the same network as SCL:
   "sensorStatus"(manualModeActive := #manualModeActive,
                  automaticModeActive := #automaticModeActive,
                  sensorActive := #sensorActive[13],
                  sensorRequested := #sensorRequested[13],
                  sensorMask := #sensorMask[13],
                  sensorStatus => #sensorStatus[13]);
END_REGION

REGION Network 15: Status 14
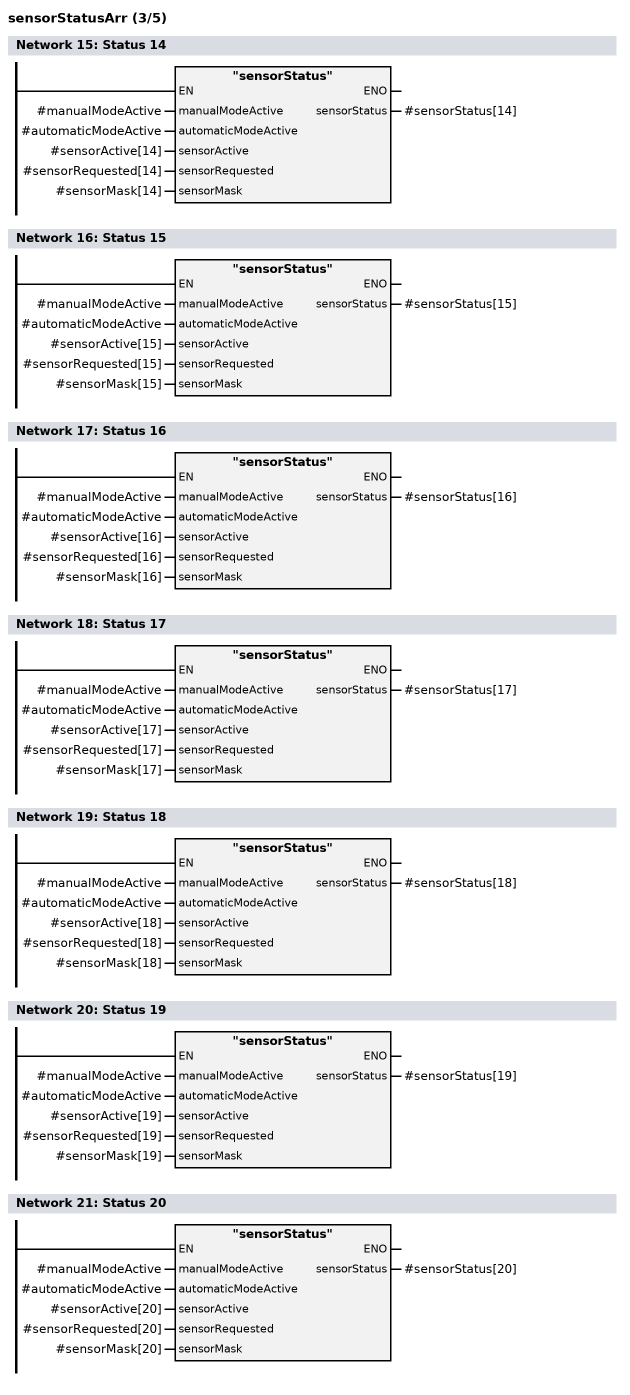
   RUNG wire#powerrail
      "sensorStatus"(manualModeActive := #manualModeActive, automaticModeActive := #automaticModeActive, sensorActive := #sensorActive[14], sensorRequested := #sensorRequested[14], sensorMask := #sensorMask[14], sensorStatus => #sensorStatus[14])
   END_RUNG
   // the same network as SCL:
   "sensorStatus"(manualModeActive := #manualModeActive,
                  automaticModeActive := #automaticModeActive,
                  sensorActive := #sensorActive[14],
                  sensorRequested := #sensorRequested[14],
                  sensorMask := #sensorMask[14],
                  sensorStatus => #sensorStatus[14]);
END_REGION

REGION Network 16: Status 15
   RUNG wire#powerrail
      "sensorStatus"(manualModeActive := #manualModeActive, automaticModeActive := #automaticModeActive, sensorActive := #sensorActive[15], sensorRequested := #sensorRequested[15], sensorMask := #sensorMask[15], sensorStatus => #sensorStatus[15])
   END_RUNG
   // the same network as SCL:
   "sensorStatus"(manualModeActive := #manualModeActive,
                  automaticModeActive := #automaticModeActive,
                  sensorActive := #sensorActive[15],
                  sensorRequested := #sensorRequested[15],
                  sensorMask := #sensorMask[15],
                  sensorStatus => #sensorStatus[15]);
END_REGION

REGION Network 17: Status 16
   RUNG wire#powerrail
      "sensorStatus"(manualModeActive := #manualModeActive, automaticModeActive := #automaticModeActive, sensorActive := #sensorActive[16], sensorRequested := #sensorRequested[16], sensorMask := #sensorMask[16], sensorStatus => #sensorStatus[16])
   END_RUNG
   // the same network as SCL:
   "sensorStatus"(manualModeActive := #manualModeActive,
                  automaticModeActive := #automaticModeActive,
                  sensorActive := #sensorActive[16],
                  sensorRequested := #sensorRequested[16],
                  sensorMask := #sensorMask[16],
                  sensorStatus => #sensorStatus[16]);
END_REGION

REGION Network 18: Status 17
   RUNG wire#powerrail
      "sensorStatus"(manualModeActive := #manualModeActive, automaticModeActive := #automaticModeActive, sensorActive := #sensorActive[17], sensorRequested := #sensorRequested[17], sensorMask := #sensorMask[17], sensorStatus => #sensorStatus[17])
   END_RUNG
   // the same network as SCL:
   "sensorStatus"(manualModeActive := #manualModeActive,
                  automaticModeActive := #automaticModeActive,
                  sensorActive := #sensorActive[17],
                  sensorRequested := #sensorRequested[17],
                  sensorMask := #sensorMask[17],
                  sensorStatus => #sensorStatus[17]);
END_REGION

REGION Network 19: Status 18
   RUNG wire#powerrail
      "sensorStatus"(manualModeActive := #manualModeActive, automaticModeActive := #automaticModeActive, sensorActive := #sensorActive[18], sensorRequested := #sensorRequested[18], sensorMask := #sensorMask[18], sensorStatus => #sensorStatus[18])
   END_RUNG
   // the same network as SCL:
   "sensorStatus"(manualModeActive := #manualModeActive,
                  automaticModeActive := #automaticModeActive,
                  sensorActive := #sensorActive[18],
                  sensorRequested := #sensorRequested[18],
                  sensorMask := #sensorMask[18],
                  sensorStatus => #sensorStatus[18]);
END_REGION

REGION Network 20: Status 19
   RUNG wire#powerrail
      "sensorStatus"(manualModeActive := #manualModeActive, automaticModeActive := #automaticModeActive, sensorActive := #sensorActive[19], sensorRequested := #sensorRequested[19], sensorMask := #sensorMask[19], sensorStatus => #sensorStatus[19])
   END_RUNG
   // the same network as SCL:
   "sensorStatus"(manualModeActive := #manualModeActive,
                  automaticModeActive := #automaticModeActive,
                  sensorActive := #sensorActive[19],
                  sensorRequested := #sensorRequested[19],
                  sensorMask := #sensorMask[19],
                  sensorStatus => #sensorStatus[19]);
END_REGION

REGION Network 21: Status 20
   RUNG wire#powerrail
      "sensorStatus"(manualModeActive := #manualModeActive, automaticModeActive := #automaticModeActive, sensorActive := #sensorActive[20], sensorRequested := #sensorRequested[20], sensorMask := #sensorMask[20], sensorStatus => #sensorStatus[20])
   END_RUNG
   // the same network as SCL:
   "sensorStatus"(manualModeActive := #manualModeActive,
                  automaticModeActive := #automaticModeActive,
                  sensorActive := #sensorActive[20],
                  sensorRequested := #sensorRequested[20],
                  sensorMask := #sensorMask[20],
                  sensorStatus => #sensorStatus[20]);
END_REGION

REGION Network 22: Status 21
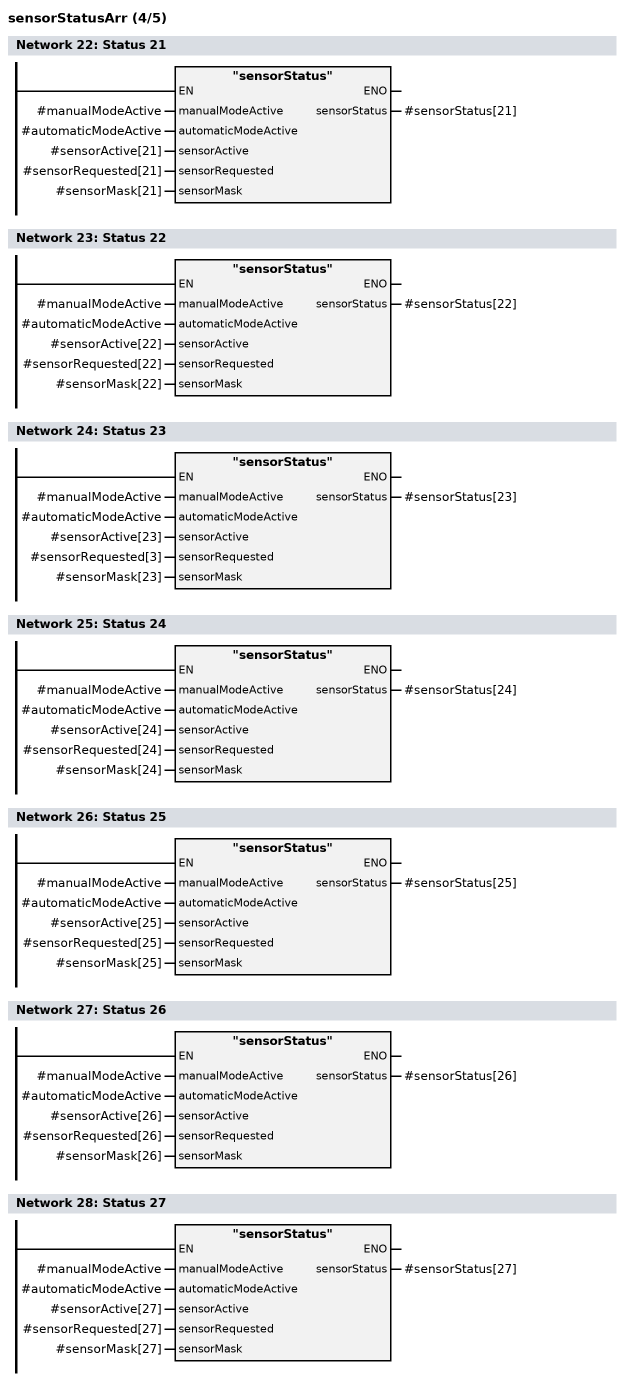
   RUNG wire#powerrail
      "sensorStatus"(manualModeActive := #manualModeActive, automaticModeActive := #automaticModeActive, sensorActive := #sensorActive[21], sensorRequested := #sensorRequested[21], sensorMask := #sensorMask[21], sensorStatus => #sensorStatus[21])
   END_RUNG
   // the same network as SCL:
   "sensorStatus"(manualModeActive := #manualModeActive,
                  automaticModeActive := #automaticModeActive,
                  sensorActive := #sensorActive[21],
                  sensorRequested := #sensorRequested[21],
                  sensorMask := #sensorMask[21],
                  sensorStatus => #sensorStatus[21]);
END_REGION

REGION Network 23: Status 22
   RUNG wire#powerrail
      "sensorStatus"(manualModeActive := #manualModeActive, automaticModeActive := #automaticModeActive, sensorActive := #sensorActive[22], sensorRequested := #sensorRequested[22], sensorMask := #sensorMask[22], sensorStatus => #sensorStatus[22])
   END_RUNG
   // the same network as SCL:
   "sensorStatus"(manualModeActive := #manualModeActive,
                  automaticModeActive := #automaticModeActive,
                  sensorActive := #sensorActive[22],
                  sensorRequested := #sensorRequested[22],
                  sensorMask := #sensorMask[22],
                  sensorStatus => #sensorStatus[22]);
END_REGION

REGION Network 24: Status 23
   RUNG wire#powerrail
      "sensorStatus"(manualModeActive := #manualModeActive, automaticModeActive := #automaticModeActive, sensorActive := #sensorActive[23], sensorRequested := #sensorRequested[3], sensorMask := #sensorMask[23], sensorStatus => #sensorStatus[23])
   END_RUNG
   // the same network as SCL:
   "sensorStatus"(manualModeActive := #manualModeActive,
                  automaticModeActive := #automaticModeActive,
                  sensorActive := #sensorActive[23],
                  sensorRequested := #sensorRequested[3],
                  sensorMask := #sensorMask[23],
                  sensorStatus => #sensorStatus[23]);
END_REGION

REGION Network 25: Status 24
   RUNG wire#powerrail
      "sensorStatus"(manualModeActive := #manualModeActive, automaticModeActive := #automaticModeActive, sensorActive := #sensorActive[24], sensorRequested := #sensorRequested[24], sensorMask := #sensorMask[24], sensorStatus => #sensorStatus[24])
   END_RUNG
   // the same network as SCL:
   "sensorStatus"(manualModeActive := #manualModeActive,
                  automaticModeActive := #automaticModeActive,
                  sensorActive := #sensorActive[24],
                  sensorRequested := #sensorRequested[24],
                  sensorMask := #sensorMask[24],
                  sensorStatus => #sensorStatus[24]);
END_REGION

REGION Network 26: Status 25
   RUNG wire#powerrail
      "sensorStatus"(manualModeActive := #manualModeActive, automaticModeActive := #automaticModeActive, sensorActive := #sensorActive[25], sensorRequested := #sensorRequested[25], sensorMask := #sensorMask[25], sensorStatus => #sensorStatus[25])
   END_RUNG
   // the same network as SCL:
   "sensorStatus"(manualModeActive := #manualModeActive,
                  automaticModeActive := #automaticModeActive,
                  sensorActive := #sensorActive[25],
                  sensorRequested := #sensorRequested[25],
                  sensorMask := #sensorMask[25],
                  sensorStatus => #sensorStatus[25]);
END_REGION

REGION Network 27: Status 26
   RUNG wire#powerrail
      "sensorStatus"(manualModeActive := #manualModeActive, automaticModeActive := #automaticModeActive, sensorActive := #sensorActive[26], sensorRequested := #sensorRequested[26], sensorMask := #sensorMask[26], sensorStatus => #sensorStatus[26])
   END_RUNG
   // the same network as SCL:
   "sensorStatus"(manualModeActive := #manualModeActive,
                  automaticModeActive := #automaticModeActive,
                  sensorActive := #sensorActive[26],
                  sensorRequested := #sensorRequested[26],
                  sensorMask := #sensorMask[26],
                  sensorStatus => #sensorStatus[26]);
END_REGION

REGION Network 28: Status 27
   RUNG wire#powerrail
      "sensorStatus"(manualModeActive := #manualModeActive, automaticModeActive := #automaticModeActive, sensorActive := #sensorActive[27], sensorRequested := #sensorRequested[27], sensorMask := #sensorMask[27], sensorStatus => #sensorStatus[27])
   END_RUNG
   // the same network as SCL:
   "sensorStatus"(manualModeActive := #manualModeActive,
                  automaticModeActive := #automaticModeActive,
                  sensorActive := #sensorActive[27],
                  sensorRequested := #sensorRequested[27],
                  sensorMask := #sensorMask[27],
                  sensorStatus => #sensorStatus[27]);
END_REGION

REGION Network 29: Status 28
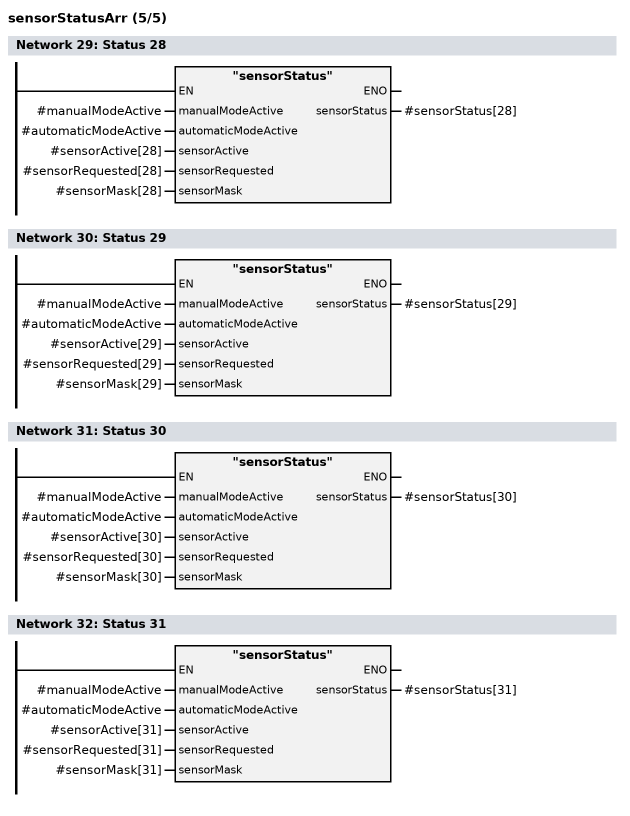
   RUNG wire#powerrail
      "sensorStatus"(manualModeActive := #manualModeActive, automaticModeActive := #automaticModeActive, sensorActive := #sensorActive[28], sensorRequested := #sensorRequested[28], sensorMask := #sensorMask[28], sensorStatus => #sensorStatus[28])
   END_RUNG
   // the same network as SCL:
   "sensorStatus"(manualModeActive := #manualModeActive,
                  automaticModeActive := #automaticModeActive,
                  sensorActive := #sensorActive[28],
                  sensorRequested := #sensorRequested[28],
                  sensorMask := #sensorMask[28],
                  sensorStatus => #sensorStatus[28]);
END_REGION

REGION Network 30: Status 29
   RUNG wire#powerrail
      "sensorStatus"(manualModeActive := #manualModeActive, automaticModeActive := #automaticModeActive, sensorActive := #sensorActive[29], sensorRequested := #sensorRequested[29], sensorMask := #sensorMask[29], sensorStatus => #sensorStatus[29])
   END_RUNG
   // the same network as SCL:
   "sensorStatus"(manualModeActive := #manualModeActive,
                  automaticModeActive := #automaticModeActive,
                  sensorActive := #sensorActive[29],
                  sensorRequested := #sensorRequested[29],
                  sensorMask := #sensorMask[29],
                  sensorStatus => #sensorStatus[29]);
END_REGION

REGION Network 31: Status 30
   RUNG wire#powerrail
      "sensorStatus"(manualModeActive := #manualModeActive, automaticModeActive := #automaticModeActive, sensorActive := #sensorActive[30], sensorRequested := #sensorRequested[30], sensorMask := #sensorMask[30], sensorStatus => #sensorStatus[30])
   END_RUNG
   // the same network as SCL:
   "sensorStatus"(manualModeActive := #manualModeActive,
                  automaticModeActive := #automaticModeActive,
                  sensorActive := #sensorActive[30],
                  sensorRequested := #sensorRequested[30],
                  sensorMask := #sensorMask[30],
                  sensorStatus => #sensorStatus[30]);
END_REGION

REGION Network 32: Status 31
   RUNG wire#powerrail
      "sensorStatus"(manualModeActive := #manualModeActive, automaticModeActive := #automaticModeActive, sensorActive := #sensorActive[31], sensorRequested := #sensorRequested[31], sensorMask := #sensorMask[31], sensorStatus => #sensorStatus[31])
   END_RUNG
   // the same network as SCL:
   "sensorStatus"(manualModeActive := #manualModeActive,
                  automaticModeActive := #automaticModeActive,
                  sensorActive := #sensorActive[31],
                  sensorRequested := #sensorRequested[31],
                  sensorMask := #sensorMask[31],
                  sensorStatus => #sensorStatus[31]);
END_REGION
END_FUNCTION

FUNCTION "torqueProfinet" : Void   // FC12, LAD
{ S7_Optimized_Access := 'TRUE' }
VERSION : 0.1
// stored: AutoNumber true, IsIECCheckEnabled false, SetENOAutomatically false, UDAEnableTagReadback false
   VAR_TEMP   // added for the SCL form of the ladder/FBD networks
      _w1 : Bool;
   END_VAR
BEGIN

REGION Network 1: HABILITAR HERRAMIENTA
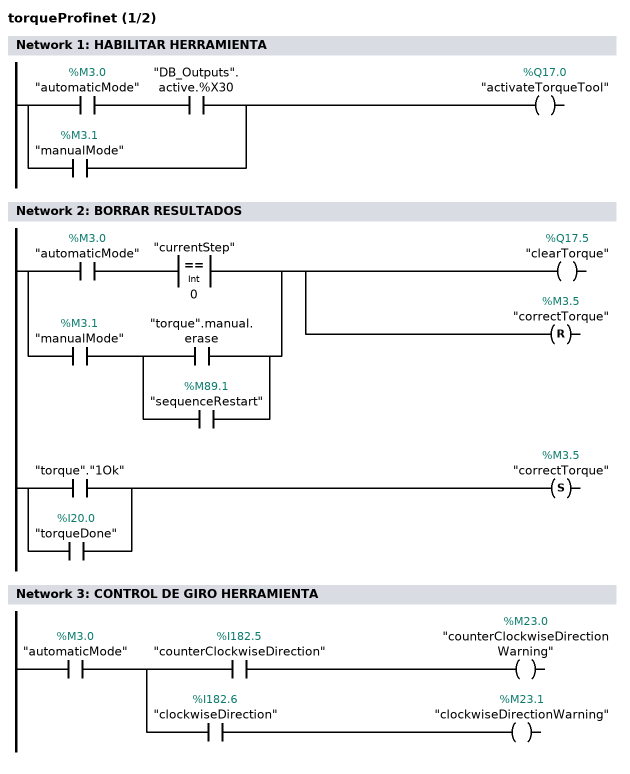
   RUNG wire#powerrail
      Contact( "automaticMode" )
      Contact( "DB_Outputs".active.%X30 )
      wire#w1
      Coil( "activateTorqueTool" )
   END_RUNG
   RUNG wire#powerrail
      Contact( "manualMode" )
   END_RUNG wire#w1
   // the same network as SCL:
   "activateTorqueTool" := ("automaticMode" AND "DB_Outputs".active.%X30) OR "manualMode";
END_REGION

REGION Network 2: BORRAR RESULTADOS
   RUNG wire#powerrail
      Contact( "automaticMode" )
      { S7_Templates := "SrcType := Int" } EQ_Contact(in1 := "currentStep", in2 := 0)
      wire#w1
      Coil( "clearTorque" )
   END_RUNG
   RUNG wire#powerrail
      Contact( "manualMode" )
      wire#w2
      Contact( "torque".manual.erase )
   END_RUNG wire#w1
   RUNG wire#w2
      Contact( "sequenceRestart" )
   END_RUNG wire#w1
   RUNG wire#w1
      R_Coil( "correctTorque" )
   END_RUNG
   RUNG wire#powerrail
      Contact( "torque"."1Ok" )
      wire#w3
      S_Coil( "correctTorque" )
   END_RUNG
   RUNG wire#powerrail
      Contact( "torqueDone" )
   END_RUNG wire#w3
   // the same network as SCL:
   "clearTorque" := ("automaticMode" AND ("currentStep" = 0)) OR ("manualMode" AND ("torque".manual.erase OR "sequenceRestart"));
   IF "clearTorque" THEN "correctTorque" := FALSE; END_IF;
   IF "torque"."1Ok" OR "torqueDone" THEN "correctTorque" := TRUE; END_IF;
END_REGION

REGION Network 3: CONTROL DE GIRO HERRAMIENTA
   RUNG wire#powerrail
      Contact( "automaticMode" )
      wire#w1
      Contact( "counterClockwiseDirection" )
      Coil( "counterClockwiseDirectionWarning" )
   END_RUNG
   RUNG wire#w1
      Contact( "clockwiseDirection" )
      Coil( "clockwiseDirectionWarning" )
   END_RUNG
   // the same network as SCL:
   "counterClockwiseDirectionWarning" := "automaticMode" AND "counterClockwiseDirection";
   "clockwiseDirectionWarning" := "automaticMode" AND "clockwiseDirection";
END_REGION

REGION Network 4: TORQUE P6000 1
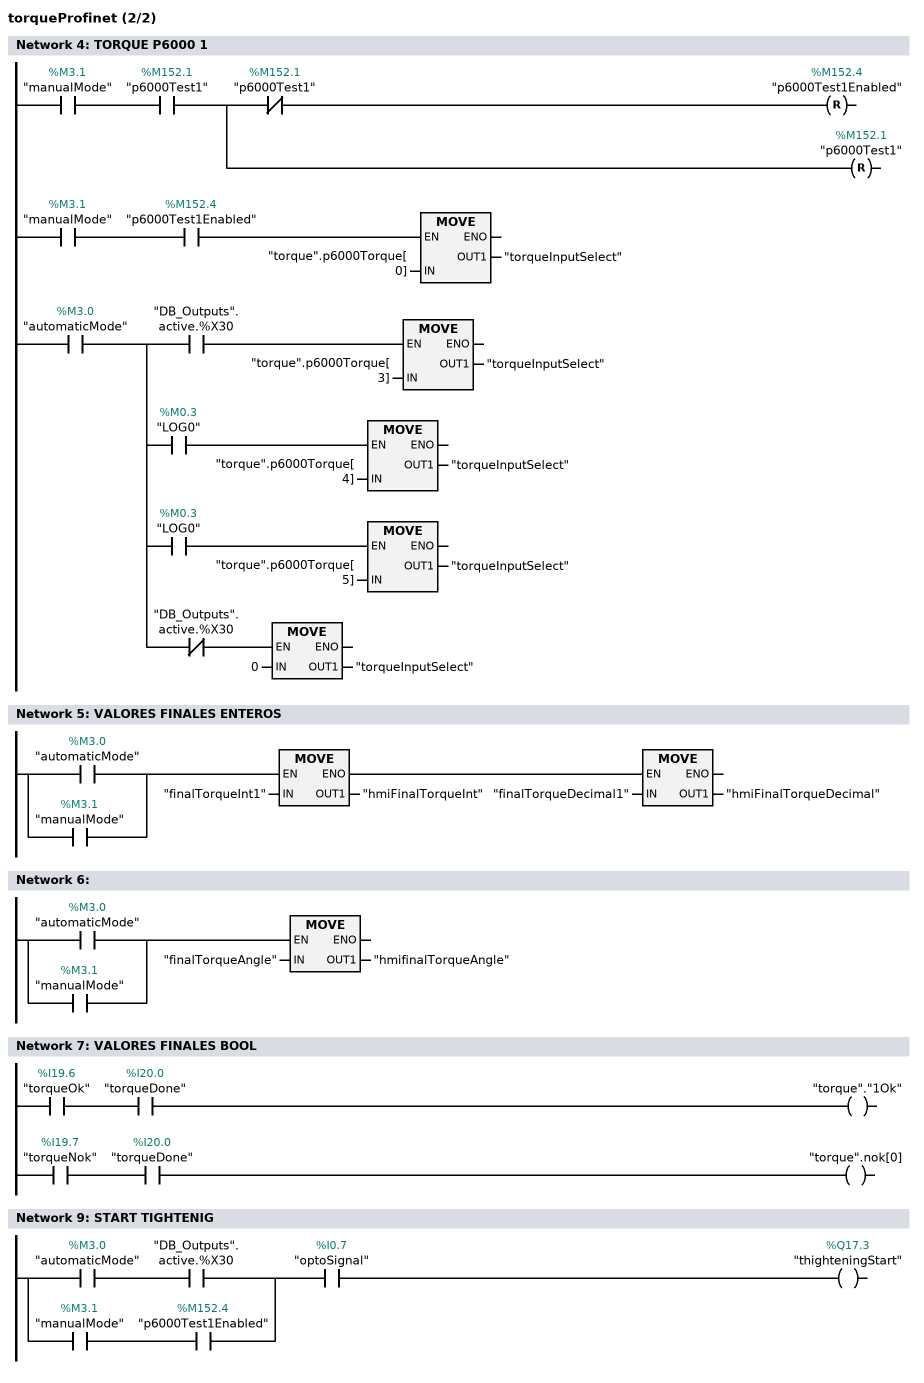
   RUNG wire#powerrail
      Contact( "manualMode" )
      Contact( "p6000Test1" )
      wire#w1
      I_Contact( "p6000Test1" )
      R_Coil( "p6000Test1Enabled" )
   END_RUNG
   RUNG wire#w1
      R_Coil( "p6000Test1" )
   END_RUNG
   RUNG wire#powerrail
      Contact( "manualMode" )
      Contact( "p6000Test1Enabled" )
      Move(in := "torque".p6000Torque[0], out1 => "torqueInputSelect")
   END_RUNG
   RUNG wire#powerrail
      Contact( "automaticMode" )
      wire#w2
      Contact( "DB_Outputs".active.%X30 )
      Move(in := "torque".p6000Torque[3], out1 => "torqueInputSelect")
   END_RUNG
   RUNG wire#w2
      Contact( "LOG0" )
      Move(in := "torque".p6000Torque[4], out1 => "torqueInputSelect")
   END_RUNG
   RUNG wire#w2
      Contact( "LOG0" )
      Move(in := "torque".p6000Torque[5], out1 => "torqueInputSelect")
   END_RUNG
   RUNG wire#w2
      I_Contact( "DB_Outputs".active.%X30 )
      Move(in := 0, out1 => "torqueInputSelect")
   END_RUNG
   // the same network as SCL:
   #_w1 := "manualMode" AND "p6000Test1";
   IF #_w1 AND NOT "p6000Test1" THEN "p6000Test1Enabled" := FALSE; END_IF;
   IF #_w1 THEN "p6000Test1" := FALSE; END_IF;
   IF "manualMode" AND "p6000Test1Enabled" THEN "torqueInputSelect" := "torque".p6000Torque[0]; END_IF;
   IF "automaticMode" AND "DB_Outputs".active.%X30 THEN
       "torqueInputSelect" := "torque".p6000Torque[3];
   END_IF;
   IF "automaticMode" AND "LOG0" THEN
       "torqueInputSelect" := "torque".p6000Torque[4];
       "torqueInputSelect" := "torque".p6000Torque[5];
   END_IF;
   IF "automaticMode" AND NOT "DB_Outputs".active.%X30 THEN "torqueInputSelect" := 0; END_IF;
END_REGION

REGION Network 5: VALORES FINALES ENTEROS
   RUNG wire#powerrail
      Contact( "automaticMode" )
      wire#w1
      Move(in := "finalTorqueInt1", out1 => "hmiFinalTorqueInt")
      Move(in := "finalTorqueDecimal1", out1 => "hmiFinalTorqueDecimal")
   END_RUNG
   RUNG wire#powerrail
      Contact( "manualMode" )
   END_RUNG wire#w1
   // the same network as SCL:
   IF "automaticMode" OR "manualMode" THEN
       "hmiFinalTorqueInt" := "finalTorqueInt1";
       "hmiFinalTorqueDecimal" := "finalTorqueDecimal1";
   END_IF;
END_REGION

REGION Network 6
   RUNG wire#powerrail
      Contact( "automaticMode" )
      wire#w1
      Move(in := "finalTorqueAngle", out1 => "hmifinalTorqueAngle")
   END_RUNG
   RUNG wire#powerrail
      Contact( "manualMode" )
   END_RUNG wire#w1
   // the same network as SCL:
   IF "automaticMode" OR "manualMode" THEN "hmifinalTorqueAngle" := "finalTorqueAngle"; END_IF;
END_REGION

REGION Network 7: VALORES FINALES BOOL
   RUNG wire#powerrail
      Contact( "torqueOk" )
      Contact( "torqueDone" )
      Coil( "torque"."1Ok" )
   END_RUNG
   RUNG wire#powerrail
      Contact( "torqueNok" )
      Contact( "torqueDone" )
      Coil( "torque".nok[0] )
   END_RUNG
   // the same network as SCL:
   "torque"."1Ok" := "torqueOk" AND "torqueDone";
   "torque".nok[0] := "torqueNok" AND "torqueDone";
END_REGION

REGION Network 8: TRS
END_REGION

REGION Network 9: START TIGHTENIG
   RUNG wire#powerrail
      Contact( "automaticMode" )
      Contact( "DB_Outputs".active.%X30 )
      wire#w1
      Contact( "optoSignal" )
      Coil( "thighteningStart" )
   END_RUNG
   RUNG wire#powerrail
      Contact( "manualMode" )
      Contact( "p6000Test1Enabled" )
   END_RUNG wire#w1
   // the same network as SCL:
   "thighteningStart" := (("automaticMode" AND "DB_Outputs".active.%X30) OR ("manualMode" AND "p6000Test1Enabled")) AND "optoSignal";
END_REGION
END_FUNCTION

FUNCTION "SCANNER CONFIG" : Void   // FC11, LAD
{ S7_Optimized_Access := 'TRUE' }
VERSION : 0.1
// stored: AutoNumber true, IsIECCheckEnabled false, SetENOAutomatically false, UDAEnableTagReadback false
   VAR_TEMP   // added for the SCL form of the ladder/FBD networks
      _w1 : Bool;
   END_VAR
BEGIN

REGION Network 1: NEST CODE READING
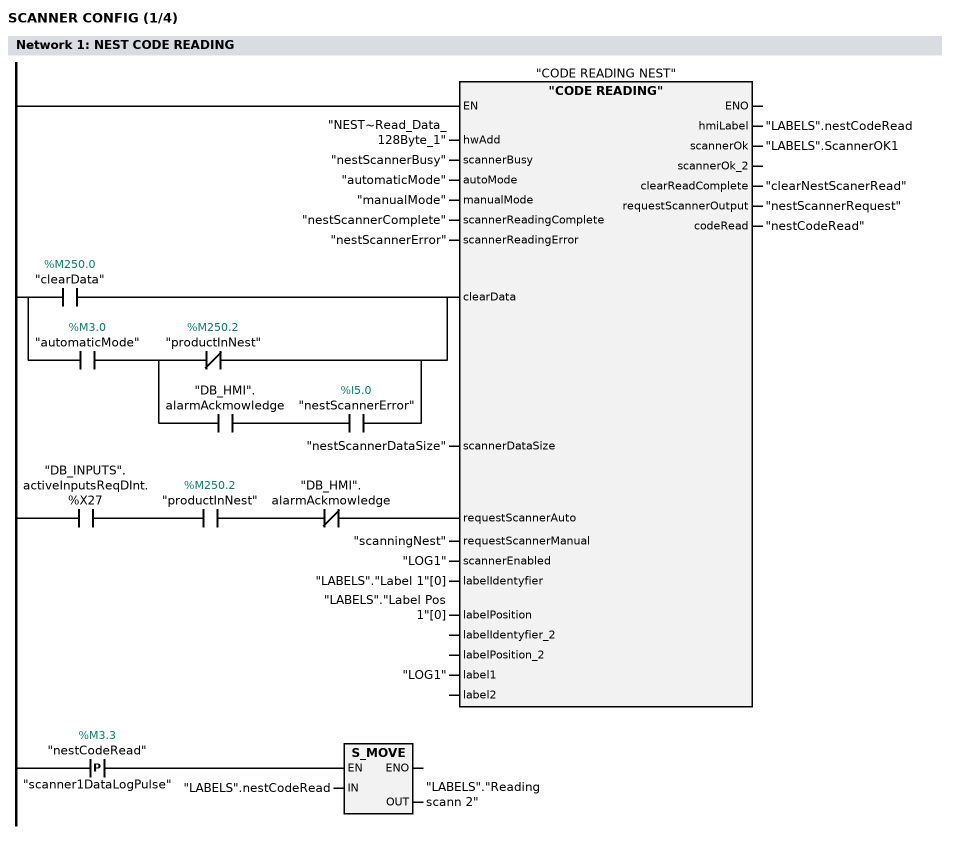
   RUNG wire#powerrail
      "CODE READING NEST"(clearData := wire#w2, requestScannerAuto := wire#w3, hwAdd := "NEST~Read_Data_128Byte_1", scannerBusy := "nestScannerBusy", autoMode := "automaticMode", manualMode := "manualMode", scannerReadingComplete := "nestScannerComplete", scannerReadingError := "nestScannerError", scannerDataSize := "nestScannerDataSize", requestScannerManual := "scanningNest", scannerEnabled := "LOG1", labelIdentyfier := "LABELS"."Label 1"[0], labelPosition := "LABELS"."Label Pos 1"[0], labelIdentyfier_2 :=, labelPosition_2 :=, label1 := "LOG1", label2 :=, hmiLabel => "LABELS".nestCodeRead, scannerOk => "LABELS".ScannerOK1, scannerOk_2 =>, clearReadComplete => "clearNestScanerRead", requestScannerOutput => "nestScannerRequest", codeRead => "nestCodeRead")
   END_RUNG
   RUNG wire#powerrail
      Contact( "clearData" )
   END_RUNG wire#w2
   RUNG wire#powerrail
      Contact( "automaticMode" )
      wire#w1
      I_Contact( "productInNest" )
   END_RUNG wire#w2
   RUNG wire#w1
      Contact( "DB_HMI".alarmAckmowledge )
      Contact( "nestScannerError" )
   END_RUNG wire#w2
   RUNG wire#powerrail
      Contact( "DB_INPUTS".activeInputsReqDInt.%X27 )
      Contact( "productInNest" )
      I_Contact( "DB_HMI".alarmAckmowledge )
   END_RUNG wire#w3
   RUNG wire#powerrail
      P_Contact(operand := "nestCodeRead", bit := "scanner1DataLogPulse")
      S_Move(in := "LABELS".nestCodeRead, out => "LABELS"."Reading scann 2")
   END_RUNG
   // the same network as SCL:
   "CODE READING NEST"(hwAdd := "NEST~Read_Data_128Byte_1",   // "CODE READING"
                       scannerBusy := "nestScannerBusy",
                       autoMode := "automaticMode",
                       manualMode := "manualMode",
                       scannerReadingComplete := "nestScannerComplete",
                       scannerReadingError := "nestScannerError",
                       clearData := "clearData" OR ("automaticMode" AND (NOT "productInNest" OR ("DB_HMI".alarmAckmowledge AND "nestScannerError"))),
                       scannerDataSize := "nestScannerDataSize",
                       requestScannerAuto := "DB_INPUTS".activeInputsReqDInt.%X27 AND "productInNest" AND NOT "DB_HMI".alarmAckmowledge,
                       requestScannerManual := "scanningNest",
                       scannerEnabled := "LOG1",
                       labelIdentyfier := "LABELS"."Label 1"[0],
                       labelPosition := "LABELS"."Label Pos 1"[0],
                       label1 := "LOG1",
                       hmiLabel => "LABELS".nestCodeRead,
                       scannerOk => "LABELS".ScannerOK1,
                       clearReadComplete => "clearNestScanerRead",
                       requestScannerOutput => "nestScannerRequest",
                       codeRead => "nestCodeRead");
   #_w1 := "nestCodeRead" AND NOT "scanner1DataLogPulse";   // rising edge of "nestCodeRead"
   "scanner1DataLogPulse" := "nestCodeRead";
   IF #_w1 THEN "LABELS"."Reading scann 2" := "LABELS".nestCodeRead; END_IF;
END_REGION

REGION Network 2: UPPER CODE READING
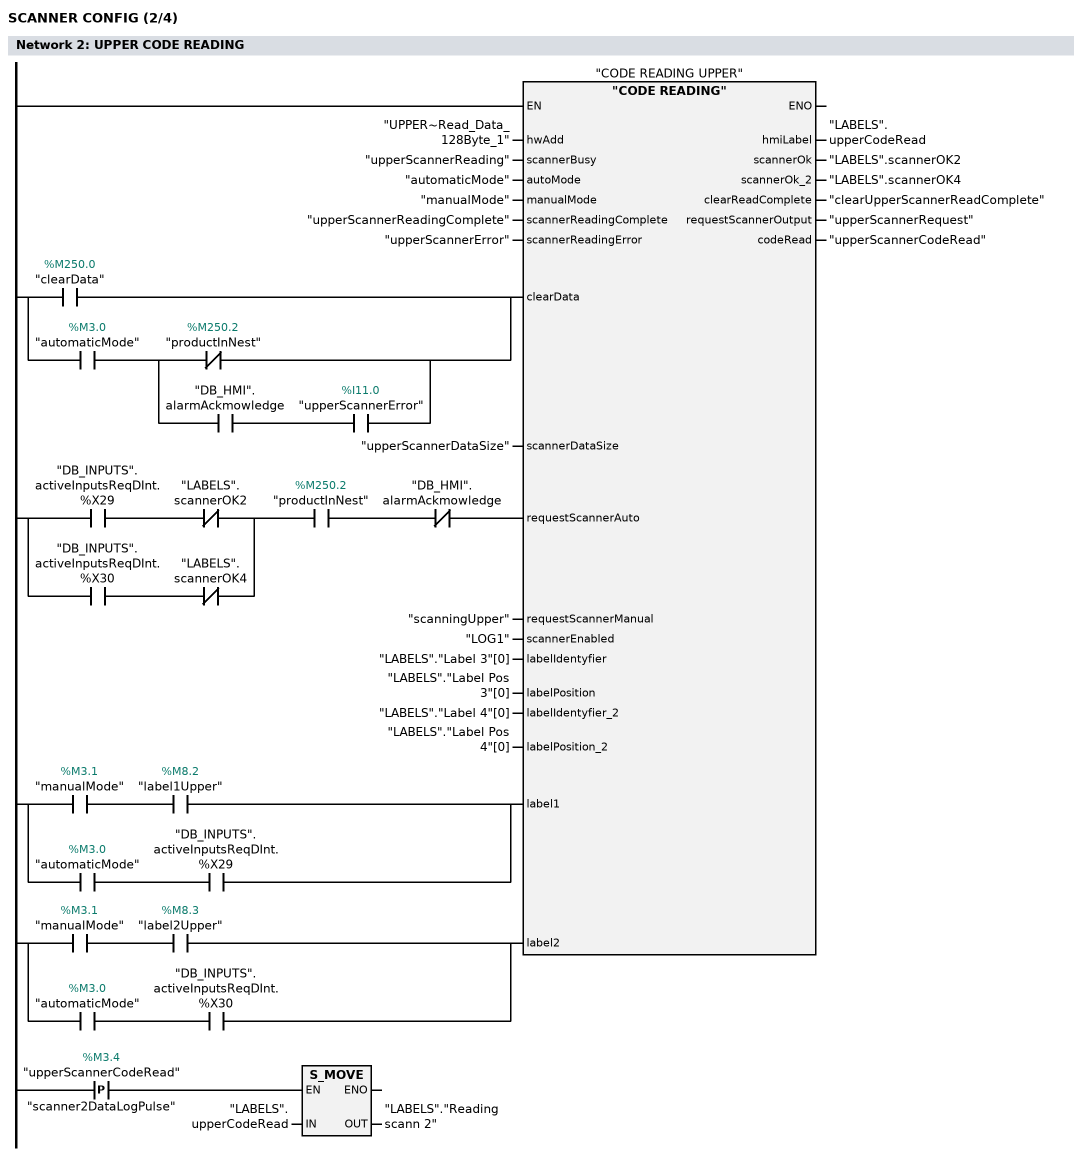
   RUNG wire#powerrail
      "CODE READING UPPER"(clearData := wire#w2, requestScannerAuto := wire#w4, label1 := wire#w5, label2 := wire#w6, hwAdd := "UPPER~Read_Data_128Byte_1", scannerBusy := "upperScannerReading", autoMode := "automaticMode", manualMode := "manualMode", scannerReadingComplete := "upperScannerReadingComplete", scannerReadingError := "upperScannerError", scannerDataSize := "upperScannerDataSize", requestScannerManual := "scanningUpper", scannerEnabled := "LOG1", labelIdentyfier := "LABELS"."Label 3"[0], labelPosition := "LABELS"."Label Pos 3"[0], labelIdentyfier_2 := "LABELS"."Label 4"[0], labelPosition_2 := "LABELS"."Label Pos 4"[0], hmiLabel => "LABELS".upperCodeRead, scannerOk => "LABELS".scannerOK2, scannerOk_2 => "LABELS".scannerOK4, clearReadComplete => "clearUpperScannerReadComplete", requestScannerOutput => "upperScannerRequest", codeRead => "upperScannerCodeRead")
   END_RUNG
   RUNG wire#powerrail
      Contact( "clearData" )
   END_RUNG wire#w2
   RUNG wire#powerrail
      Contact( "automaticMode" )
      wire#w1
      I_Contact( "productInNest" )
   END_RUNG wire#w2
   RUNG wire#w1
      Contact( "DB_HMI".alarmAckmowledge )
      Contact( "upperScannerError" )
   END_RUNG wire#w2
   RUNG wire#powerrail
      Contact( "DB_INPUTS".activeInputsReqDInt.%X29 )
      I_Contact( "LABELS".scannerOK2 )
      wire#w3
      Contact( "productInNest" )
      I_Contact( "DB_HMI".alarmAckmowledge )
   END_RUNG wire#w4
   RUNG wire#powerrail
      Contact( "DB_INPUTS".activeInputsReqDInt.%X30 )
      I_Contact( "LABELS".scannerOK4 )
   END_RUNG wire#w3
   RUNG wire#powerrail
      Contact( "manualMode" )
      Contact( "label1Upper" )
   END_RUNG wire#w5
   RUNG wire#powerrail
      Contact( "automaticMode" )
      Contact( "DB_INPUTS".activeInputsReqDInt.%X29 )
   END_RUNG wire#w5
   RUNG wire#powerrail
      Contact( "manualMode" )
      Contact( "label2Upper" )
   END_RUNG wire#w6
   RUNG wire#powerrail
      Contact( "automaticMode" )
      Contact( "DB_INPUTS".activeInputsReqDInt.%X30 )
   END_RUNG wire#w6
   RUNG wire#powerrail
      P_Contact(operand := "upperScannerCodeRead", bit := "scanner2DataLogPulse")
      S_Move(in := "LABELS".upperCodeRead, out => "LABELS"."Reading scann 2")
   END_RUNG
   // the same network as SCL:
   "CODE READING UPPER"(hwAdd := "UPPER~Read_Data_128Byte_1",   // "CODE READING"
                        scannerBusy := "upperScannerReading",
                        autoMode := "automaticMode",
                        manualMode := "manualMode",
                        scannerReadingComplete := "upperScannerReadingComplete",
                        scannerReadingError := "upperScannerError",
                        clearData := "clearData" OR ("automaticMode" AND (NOT "productInNest" OR ("DB_HMI".alarmAckmowledge AND "upperScannerError"))),
                        scannerDataSize := "upperScannerDataSize",
                        requestScannerAuto := (("DB_INPUTS".activeInputsReqDInt.%X29 AND NOT "LABELS".scannerOK2) OR ("DB_INPUTS".activeInputsReqDInt.%X30 AND NOT "LABELS".scannerOK4)) AND "productInNest" AND NOT "DB_HMI".alarmAckmowledge,
                        requestScannerManual := "scanningUpper",
                        scannerEnabled := "LOG1",
                        labelIdentyfier := "LABELS"."Label 3"[0],
                        labelPosition := "LABELS"."Label Pos 3"[0],
                        labelIdentyfier_2 := "LABELS"."Label 4"[0],
                        labelPosition_2 := "LABELS"."Label Pos 4"[0],
                        label1 := ("manualMode" AND "label1Upper") OR ("automaticMode" AND "DB_INPUTS".activeInputsReqDInt.%X29),
                        label2 := ("manualMode" AND "label2Upper") OR ("automaticMode" AND "DB_INPUTS".activeInputsReqDInt.%X30),
                        hmiLabel => "LABELS".upperCodeRead,
                        scannerOk => "LABELS".scannerOK2,
                        scannerOk_2 => "LABELS".scannerOK4,
                        clearReadComplete => "clearUpperScannerReadComplete",
                        requestScannerOutput => "upperScannerRequest",
                        codeRead => "upperScannerCodeRead");
   #_w1 := "upperScannerCodeRead" AND NOT "scanner2DataLogPulse";   // rising edge of "upperScannerCodeRead"
   "scanner2DataLogPulse" := "upperScannerCodeRead";
   IF #_w1 THEN "LABELS"."Reading scann 2" := "LABELS".upperCodeRead; END_IF;
END_REGION

